LIN {X -0.205,Y -555.841,Z 989.032,A 0.000,B 0.000,C 90.000,E1 41.757} C_DIS
LIN {X 0.302,Y -553.942,Z 989.029,A 0.000,B 0.000,C 90.000,E1 41.148} C_DIS
LIN {X 0.015,Y -551.893,Z 989.026,A 0.000,B 0.000,C 90.000,E1 40.620} C_DIS
LIN {X -0.229,Y -548.482,Z 989.021,A 0.000,B 0.000,C 90.000,E1 39.806} C_DIS
LIN {X 0.068,Y -545.367,Z 989.017,A 0.000,B 0.000,C 90.000,E1 39.072} C_DIS
LIN {X -0.279,Y -542.695,Z 989.014,A 0.000,B 0.000,C 90.000,E1 38.543} C_DIS
LIN {X -0.021,Y -537.799,Z 989.008,A 0.000,B 0.000,C 90.000,E1 37.523} C_DIS
LIN {X 0.164,Y -534.006,Z 989.005,A 0.000,B 0.000,C 90.000,E1 36.790} C_DIS
LIN {X -0.018,Y -528.523,Z 988.999,A 0.000,B 0.000,C 90.000,E1 35.804} C_DIS
LIN {X -0.096,Y -523.405,Z 988.994,A 0.000,B 0.000,C 90.000,E1 34.945} C_DIS
LIN {X -0.098,Y -517.896,Z 988.989,A 0.000,B 0.000,C 90.000,E1 34.072} C_DIS
LIN {X 0.309,Y -513.063,Z 988.985,A 0.000,B 0.000,C 90.000,E1 33.293} C_DIS
LIN {X -0.136,Y -508.884,Z 988.982,A 0.000,B 0.000,C 90.000,E1 32.752} C_DIS
LIN {X 0.093,Y -504.403,Z 988.979,A 0.000,B 0.000,C 90.000,E1 32.133} C_DIS
LIN {X 0.215,Y -500.887,Z 988.976,A 0.000,B 0.000,C 90.000,E1 31.671} C_DIS
LIN {X -0.110,Y -497.223,Z 988.974,A 0.000,B 0.000,C 90.000,E1 31.258} C_DIS
LIN {X -0.112,Y -490.581,Z 988.969,A 0.000,B 0.000,C 90.000,E1 30.512} C_DIS
LIN {X 0.017,Y -485.022,Z 988.966,A 0.000,B 0.000,C 90.000,E1 29.922} C_DIS
LIN {X 0.172,Y -476.755,Z 988.962,A 0.000,B 0.000,C 90.000,E1 29.077} C_DIS
LIN {X -0.018,Y -470.857,Z 988.959,A 0.000,B 0.000,C 90.000,E1 28.537} C_DIS
LIN {X 0.163,Y -462.229,Z 988.954,A 0.000,B 0.000,C 90.000,E1 27.719} C_DIS
LIN {X -0.046,Y -451.758,Z 988.949,A 0.000,B 0.000,C 90.000,E1 26.821} C_DIS
LIN {X 0.042,Y -441.003,Z 988.944,A 0.000,B 0.000,C 90.000,E1 25.899} C_DIS
LIN {X 0.055,Y -420.137,Z 988.934,A 0.000,B 0.000,C 90.000,E1 24.027} C_DIS
LIN {X 0.018,Y -404.044,Z 988.925,A 0.000,B 0.000,C 90.000,E1 22.408} C_DIS
LIN {X -0.078,Y -399.969,Z 988.922,A 0.000,B 0.000,C 90.000,E1 21.972} C_DIS
LIN {X -0.199,Y -397.751,Z 988.921,A 0.000,B 0.000,C 90.000,E1 21.716} C_DIS
LIN {X 0.151,Y -393.382,Z 988.917,A 0.000,B 0.000,C 90.000,E1 21.046} C_DIS
LIN {X -0.105,Y -391.732,Z 988.915,A 0.000,B 0.000,C 90.000,E1 20.737} C_DIS
LIN {X 0.033,Y -390.332,Z 988.912,A 0.000,B 0.000,C 90.000,E1 20.066} C_DIS
LIN {X 0.090,Y -390.055,Z 988.908,A 0.000,B 0.000,C 90.000,E1 19.504} C_DIS
LIN {X -0.118,Y -390.561,Z 988.903,A 0.000,B 0.000,C 90.000,E1 18.471} C_DIS
LIN {X 0.071,Y -393.854,Z 988.885,A 0.000,B 0.000,C 90.000,E1 15.245} C_DIS
LIN {X 0.041,Y -398.839,Z 988.863,A 0.000,B 0.000,C 90.000,E1 11.366} C_DIS
LIN {X 0.012,Y -403.989,Z 988.846,A 0.000,B 0.000,C 90.000,E1 8.219} C_DIS
LIN {X -0.049,Y -408.655,Z 988.832,A 0.000,B 0.000,C 90.000,E1 5.796} C_DIS
LIN {X -0.025,Y -414.498,Z 988.817,A 0.000,B 0.000,C 90.000,E1 3.037} C_DIS
LIN {X 0.032,Y -417.458,Z 988.809,A 0.000,B 0.000,C 90.000,E1 1.661} C_DIS
LIN {X 0.073,Y -419.347,Z 988.806,A 0.000,B 0.000,C 90.000,E1 0.974} C_DIS
LIN {X 0.087,Y -419.875,Z 988.805,A 0.000,B 0.000,C 90.000,E1 0.802} C_DIS
LIN {X -0.145,Y -422.853,Z 988.801,A 0.000,B 0.000,C 90.000,E1 0.172} C_DIS
LIN {X 0.000,Y -423.890,Z 988.800,A 0.000,B 0.000,C 90.000,E1 360.000} C_DIS
LIN {X 0.037,Y -428.403,Z 988.797,A 0.000,B 0.000,C 90.000,E1 359.484} C_DIS
LIN {X -0.134,Y -429.256,Z 988.797,A 0.000,B 0.000,C 90.000,E1 359.427} C_DIS
LIN {X -0.068,Y -433.129,Z 988.795,A 0.000,B 0.000,C 90.000,E1 359.141} C_DIS
LIN {X -0.176,Y -441.347,Z 988.793,A 0.000,B 0.000,C 90.000,E1 358.682} C_DIS
LIN {X 0.178,Y -447.909,Z 988.791,A 0.000,B 0.000,C 90.000,E1 358.282} C_DIS
LIN {X -0.169,Y -463.031,Z 988.786,A 0.000,B 0.000,C 90.000,E1 357.478} C_DIS
LIN {X 0.080,Y -474.728,Z 988.782,A 0.000,B 0.000,C 90.000,E1 356.788} C_DIS
LIN {X 0.125,Y -487.806,Z 988.778,A 0.000,B 0.000,C 90.000,E1 356.045} C_DIS
LIN {X 0.088,Y -497.730,Z 988.775,A 0.000,B 0.000,C 90.000,E1 355.469} C_DIS
LIN {X 0.097,Y -508.908,Z 988.771,A 0.000,B 0.000,C 90.000,E1 354.780} C_DIS
LIN {X 0.239,Y -518.180,Z 988.768,A 0.000,B 0.000,C 90.000,E1 354.147} C_DIS
LIN {X -0.013,Y -524.340,Z 988.765,A 0.000,B 0.000,C 90.000,E1 353.742} C_DIS
LIN {X -0.005,Y -533.163,Z 988.761,A 0.000,B 0.000,C 90.000,E1 353.053} C_DIS
LIN {X -0.120,Y -538.896,Z 988.759,A 0.000,B 0.000,C 90.000,E1 352.591} C_DIS
LIN {X -0.208,Y -546.921,Z 988.755,A 0.000,B 0.000,C 90.000,E1 351.837} C_DIS
LIN {X -0.216,Y -552.120,Z 988.752,A 0.000,B 0.000,C 90.000,E1 351.310} C_DIS
LIN {X 0.053,Y -557.053,Z 988.749,A 0.000,B 0.000,C 90.000,E1 350.735} C_DIS
LIN {X 0.076,Y -562.660,Z 988.745,A 0.000,B 0.000,C 90.000,E1 350.038} C_DIS
LIN {X -0.162,Y -566.786,Z 988.742,A 0.000,B 0.000,C 90.000,E1 349.511} C_DIS
LIN {X 0.189,Y -570.569,Z 988.739,A 0.000,B 0.000,C 90.000,E1 348.926} C_DIS
LIN {X -0.228,Y -574.843,Z 988.735,A 0.000,B 0.000,C 90.000,E1 348.285} C_DIS
LIN {X 0.183,Y -578.041,Z 988.732,A 0.000,B 0.000,C 90.000,E1 347.701} C_DIS
LIN {X -0.056,Y -583.941,Z 988.726,A 0.000,B 0.000,C 90.000,E1 346.645} C_DIS
LIN {X -0.078,Y -589.375,Z 988.720,A 0.000,B 0.000,C 90.000,E1 345.574} C_DIS
LIN {X 0.129,Y -593.291,Z 988.715,A 0.000,B 0.000,C 90.000,E1 344.755} C_DIS
LIN {X -0.054,Y -599.436,Z 988.708,A 0.000,B 0.000,C 90.000,E1 343.449} C_DIS
LIN {X -0.221,Y -603.429,Z 988.703,A 0.000,B 0.000,C 90.000,E1 342.543} C_DIS
LIN {X -0.073,Y -608.844,Z 988.696,A 0.000,B 0.000,C 90.000,E1 341.221} C_DIS
LIN {X -0.157,Y -612.837,Z 988.690,A 0.000,B 0.000,C 90.000,E1 340.188} C_DIS
LIN {X 0.065,Y -615.611,Z 988.686,A 0.000,B 0.000,C 90.000,E1 339.390} C_DIS
LIN {X 0.045,Y -619.912,Z 988.678,A 0.000,B 0.000,C 90.000,E1 338.103} C_DIS
LIN {X -0.222,Y -621.511,Z 988.676,A 0.000,B 0.000,C 90.000,E1 337.614} C_DIS
LIN {X 0.083,Y -624.635,Z 988.670,A 0.000,B 0.000,C 90.000,E1 336.561} C_DIS
LIN {X 0.131,Y -628.204,Z 988.663,A 0.000,B 0.000,C 90.000,E1 335.281} C_DIS
LIN {X -0.046,Y -630.871,Z 988.657,A 0.000,B 0.000,C 90.000,E1 334.280} C_DIS
LIN {X 0.082,Y -633.281,Z 988.651,A 0.000,B 0.000,C 90.000,E1 333.256} C_DIS
LIN {X 0.242,Y -635.421,Z 988.646,A 0.000,B 0.000,C 90.000,E1 332.231} C_DIS
LIN {X -0.088,Y -637.969,Z 988.639,A 0.000,B 0.000,C 90.000,E1 331.001} C_DIS
LIN {X -0.015,Y -640.741,Z 988.631,A 0.000,B 0.000,C 90.000,E1 329.488} C_DIS
LIN {X -0.014,Y -642.383,Z 988.625,A 0.000,B 0.000,C 90.000,E1 328.486} C_DIS
LIN {X 0.351,Y -643.812,Z 988.619,A 0.000,B 0.000,C 90.000,E1 327.454} C_DIS
LIN {X -0.148,Y -645.119,Z 988.614,A 0.000,B 0.000,C 90.000,E1 326.501} C_DIS
LIN {X 0.204,Y -645.949,Z 988.610,A 0.000,B 0.000,C 90.000,E1 325.722} C_DIS
LIN {X 0.150,Y -647.051,Z 988.603,A 0.000,B 0.000,C 90.000,E1 324.482} C_DIS
LIN {X -0.038,Y -647.948,Z 988.596,A 0.000,B 0.000,C 90.000,E1 323.256} C_DIS
LIN {X -0.127,Y -648.450,Z 988.590,A 0.000,B 0.000,C 90.000,E1 322.271} C_DIS
LIN {X 0.062,Y -649.212,Z 988.581,A 0.000,B 0.000,C 90.000,E1 320.517} C_DIS
LIN {X -0.185,Y -649.707,Z 988.574,A 0.000,B 0.000,C 90.000,E1 319.299} C_DIS
LIN {X 0.217,Y -651.382,Z 988.559,A 0.000,B 0.000,C 90.000,E1 316.539} C_DIS
LIN {X -0.070,Y -652.394,Z 988.550,A 0.000,B 0.000,C 90.000,E1 315.081} C_DIS
LIN {X 0.052,Y -653.888,Z 988.539,A 0.000,B 0.000,C 90.000,E1 313.095} C_DIS
LIN {X 0.327,Y -654.830,Z 988.533,A 0.000,B 0.000,C 90.000,E1 311.838} C_DIS
LIN {X 0.131,Y -655.799,Z 988.524,A 0.000,B 0.000,C 90.000,E1 310.378} C_DIS
LIN {X 0.076,Y -656.458,Z 988.518,A 0.000,B 0.000,C 90.000,E1 309.152} C_DIS
LIN {X -0.064,Y -657.014,Z 988.511,A 0.000,B 0.000,C 90.000,E1 307.935} C_DIS
LIN {X -0.038,Y -657.427,Z 988.505,A 0.000,B 0.000,C 90.000,E1 306.950} C_DIS
LIN {X -0.078,Y -657.603,Z 988.501,A 0.000,B 0.000,C 90.000,E1 306.217} C_DIS
LIN {X -0.020,Y -657.818,Z 988.493,A 0.000,B 0.000,C 90.000,E1 304.739} C_DIS
LIN {X 0.219,Y -658.163,Z 988.485,A 0.000,B 0.000,C 90.000,E1 303.245} C_DIS
LIN {X -0.153,Y -664.391,Z 988.448,A 0.000,B 0.000,C 90.000,E1 296.668} C_DIS
LIN {X -0.160,Y -666.765,Z 988.440,A 0.000,B 0.000,C 90.000,E1 295.207} C_DIS
LIN {X 0.175,Y -668.283,Z 988.435,A 0.000,B 0.000,C 90.000,E1 294.207} C_DIS
LIN {X -0.080,Y -669.644,Z 988.429,A 0.000,B 0.000,C 90.000,E1 293.259} C_DIS
LIN {X 0.132,Y -670.406,Z 988.425,A 0.000,B 0.000,C 90.000,E1 292.514} C_DIS
LIN {X 0.194,Y -670.504,Z 988.422,A 0.000,B 0.000,C 90.000,E1 292.025} C_DIS
LIN {X 0.102,Y -670.488,Z 988.421,A 0.000,B 0.000,C 90.000,E1 291.791} C_DIS
LIN {X -0.209,Y -669.817,Z 988.418,A 0.000,B 0.000,C 90.000,E1 291.334} C_DIS
LIN {X -0.299,Y -669.269,Z 988.417,A 0.000,B 0.000,C 90.000,E1 291.099} C_DIS
LIN {X -0.312,Y -667.339,Z 988.415,A 0.000,B 0.000,C 90.000,E1 290.737} C_DIS
LIN {X -0.168,Y -665.582,Z 988.414,A 0.000,B 0.000,C 90.000,E1 290.482} C_DIS
LIN {X -0.099,Y -664.567,Z 988.413,A 0.000,B 0.000,C 90.000,E1 290.355} C_DIS
LIN {X -0.263,Y -663.070,Z 988.412,A 0.000,B 0.000,C 90.000,E1 290.248} C_DIS
LIN {X -0.159,Y -657.023,Z 988.410,A 0.000,B 0.000,C 90.000,E1 289.812} C_DIS
LIN {X 0.031,Y -646.511,Z 988.406,A 0.000,B 0.000,C 90.000,E1 289.141} C_DIS
LIN {X -0.299,Y -645.482,Z 988.406,A 0.000,B 0.000,C 90.000,E1 289.033} C_DIS
LIN {X -0.137,Y -645.465,Z 988.406,A 0.000,B 0.000,C 90.000,E1 289.014} C_DIS
LIN {X 0.311,Y -645.574,Z 988.405,A 0.000,B 0.000,C 90.000,E1 288.779} C_DIS
LIN {X 0.096,Y -647.600,Z 988.402,A 0.000,B 0.000,C 90.000,E1 288.362} C_DIS
LIN {X -0.194,Y -655.116,Z 988.395,A 0.000,B 0.000,C 90.000,E1 287.149} C_DIS
LIN {X 0.197,Y -657.838,Z 988.393,A 0.000,B 0.000,C 90.000,E1 286.622} C_DIS
LIN {X 0.165,Y -660.338,Z 988.390,A 0.000,B 0.000,C 90.000,E1 286.134} C_DIS
LIN {X -0.040,Y -662.472,Z 988.387,A 0.000,B 0.000,C 90.000,E1 285.662} C_DIS
LIN {X -0.229,Y -664.064,Z 988.384,A 0.000,B 0.000,C 90.000,E1 285.190} C_DIS
LIN {X -0.319,Y -664.799,Z 988.383,A 0.000,B 0.000,C 90.000,E1 284.954} C_DIS
LIN {X 0.155,Y -665.943,Z 988.380,A 0.000,B 0.000,C 90.000,E1 284.426} C_DIS
LIN {X 0.074,Y -667.201,Z 988.376,A 0.000,B 0.000,C 90.000,E1 283.703} C_DIS
LIN {X -0.237,Y -667.836,Z 988.374,A 0.000,B 0.000,C 90.000,E1 283.244} C_DIS
LIN {X 0.190,Y -668.351,Z 988.369,A 0.000,B 0.000,C 90.000,E1 282.479} C_DIS
LIN {X 0.042,Y -668.507,Z 988.367,A 0.000,B 0.000,C 90.000,E1 282.007} C_DIS
LIN {X -0.185,Y -668.277,Z 988.363,A 0.000,B 0.000,C 90.000,E1 281.299} C_DIS
LIN {X 0.188,Y -667.968,Z 988.360,A 0.000,B 0.000,C 90.000,E1 280.782} C_DIS
LIN {X 0.031,Y -667.399,Z 988.357,A 0.000,B 0.000,C 90.000,E1 280.310} C_DIS
LIN {X -0.251,Y -666.652,Z 988.355,A 0.000,B 0.000,C 90.000,E1 279.849} C_DIS
LIN {X 0.037,Y -664.846,Z 988.351,A 0.000,B 0.000,C 90.000,E1 279.095} C_DIS
LIN {X -0.151,Y -663.378,Z 988.348,A 0.000,B 0.000,C 90.000,E1 278.624} C_DIS
LIN {X 0.205,Y -661.559,Z 988.345,A 0.000,B 0.000,C 90.000,E1 278.106} C_DIS
LIN {X -0.102,Y -659.443,Z 988.342,A 0.000,B 0.000,C 90.000,E1 277.644} C_DIS
LIN {X 0.126,Y -656.103,Z 988.339,A 0.000,B 0.000,C 90.000,E1 277.011} C_DIS
LIN {X -0.140,Y -652.943,Z 988.336,A 0.000,B 0.000,C 90.000,E1 276.543} C_DIS
LIN {X 0.073,Y -649.275,Z 988.334,A 0.000,B 0.000,C 90.000,E1 276.030} C_DIS
LIN {X 0.279,Y -644.043,Z 988.330,A 0.000,B 0.000,C 90.000,E1 275.391} C_DIS
LIN {X -0.198,Y -639.512,Z 988.327,A 0.000,B 0.000,C 90.000,E1 274.935} C_DIS
LIN {X 0.069,Y -634.547,Z 988.325,A 0.000,B 0.000,C 90.000,E1 274.416} C_DIS
LIN {X -0.142,Y -627.856,Z 988.321,A 0.000,B 0.000,C 90.000,E1 273.841} C_DIS
LIN {X 0.038,Y -620.746,Z 988.318,A 0.000,B 0.000,C 90.000,E1 273.269} C_DIS
LIN {X 0.278,Y -618.053,Z 988.317,A 0.000,B 0.000,C 90.000,E1 273.037} C_DIS
LIN {X -0.294,Y -610.196,Z 988.314,A 0.000,B 0.000,C 90.000,E1 272.579} C_DIS
LIN {X -0.059,Y -603.897,Z 988.312,A 0.000,B 0.000,C 90.000,E1 272.178} C_DIS
LIN {X -0.076,Y -597.093,Z 988.310,A 0.000,B 0.000,C 90.000,E1 271.835} C_DIS
LIN {X -0.072,Y -591.854,Z 988.309,A 0.000,B 0.000,C 90.000,E1 271.604} C_DIS
LIN {X 0.033,Y -584.596,Z 988.307,A 0.000,B 0.000,C 90.000,E1 271.318} C_DIS
LIN {X -0.086,Y -576.828,Z 988.306,A 0.000,B 0.000,C 90.000,E1 271.088} C_DIS
LIN {X 0.171,Y -571.043,Z 988.305,A 0.000,B 0.000,C 90.000,E1 270.917} C_DIS
LIN {X 0.168,Y -565.048,Z 988.305,A 0.000,B 0.000,C 90.000,E1 270.802} C_DIS
LIN {X -0.005,Y -558.040,Z 988.304,A 0.000,B 0.000,C 90.000,E1 270.745} C_DIS
LIN {X -0.054,Y -543.065,Z 988.304,A 0.000,B 0.000,C 90.000,E1 270.745} C_DIS
LIN {X 0.222,Y -542.570,Z 988.302,A 0.000,B 0.000,C 90.000,E1 270.401} C_DIS
LIN {X -0.025,Y -541.364,Z 988.293,A 0.000,B 0.000,C 90.000,E1 268.740} C_DIS
LIN {X 0.103,Y -540.430,Z 988.285,A 0.000,B 0.000,C 90.000,E1 267.306} C_DIS
LIN {X -0.272,Y -538.995,Z 988.274,A 0.000,B 0.000,C 90.000,E1 265.355} C_DIS
LIN {X -0.104,Y -537.811,Z 988.266,A 0.000,B 0.000,C 90.000,E1 263.913} C_DIS
LIN {X -0.005,Y -536.805,Z 988.260,A 0.000,B 0.000,C 90.000,E1 262.761} C_DIS
LIN {X 0.146,Y -535.665,Z 988.253,A 0.000,B 0.000,C 90.000,E1 261.602} C_DIS
LIN {X -0.233,Y -533.936,Z 988.244,A 0.000,B 0.000,C 90.000,E1 259.926} C_DIS
LIN {X 0.053,Y -532.092,Z 988.234,A 0.000,B 0.000,C 90.000,E1 258.173} C_DIS
LIN {X -0.181,Y -530.829,Z 988.228,A 0.000,B 0.000,C 90.000,E1 257.048} C_DIS
LIN {X 0.159,Y -528.779,Z 988.218,A 0.000,B 0.000,C 90.000,E1 255.283} C_DIS
LIN {X 0.245,Y -526.301,Z 988.206,A 0.000,B 0.000,C 90.000,E1 252.960} C_DIS
LIN {X 0.083,Y -524.969,Z 988.199,A 0.000,B 0.000,C 90.000,E1 251.819} C_DIS
LIN {X -0.102,Y -523.557,Z 988.193,A 0.000,B 0.000,C 90.000,E1 250.678} C_DIS
LIN {X 0.175,Y -521.330,Z 988.183,A 0.000,B 0.000,C 90.000,E1 248.901} C_DIS
LIN {X -0.084,Y -519.055,Z 988.173,A 0.000,B 0.000,C 90.000,E1 247.177} C_DIS
LIN {X 0.004,Y -517.409,Z 988.167,A 0.000,B 0.000,C 90.000,E1 245.997} C_DIS
LIN {X -0.190,Y -515.692,Z 988.160,A 0.000,B 0.000,C 90.000,E1 244.845} C_DIS
LIN {X -0.279,Y -513.326,Z 988.152,A 0.000,B 0.000,C 90.000,E1 243.384} C_DIS
LIN {X 0.168,Y -511.491,Z 988.145,A 0.000,B 0.000,C 90.000,E1 242.153} C_DIS
LIN {X -0.220,Y -509.066,Z 988.137,A 0.000,B 0.000,C 90.000,E1 240.717} C_DIS
LIN {X 0.080,Y -507.515,Z 988.132,A 0.000,B 0.000,C 90.000,E1 239.793} C_DIS
LIN {X -0.130,Y -504.779,Z 988.124,A 0.000,B 0.000,C 90.000,E1 238.329} C_DIS
LIN {X -0.127,Y -501.673,Z 988.116,A 0.000,B 0.000,C 90.000,E1 236.834} C_DIS
LIN {X 0.093,Y -498.396,Z 988.107,A 0.000,B 0.000,C 90.000,E1 235.308} C_DIS
LIN {X 0.112,Y -496.271,Z 988.102,A 0.000,B 0.000,C 90.000,E1 234.402} C_DIS
LIN {X -0.182,Y -492.695,Z 988.094,A 0.000,B 0.000,C 90.000,E1 232.924} C_DIS
LIN {X -0.105,Y -488.346,Z 988.084,A 0.000,B 0.000,C 90.000,E1 231.090} C_DIS
LIN {X 0.138,Y -482.608,Z 988.070,A 0.000,B 0.000,C 90.000,E1 228.609} C_DIS
LIN {X 0.272,Y -476.521,Z 988.055,A 0.000,B 0.000,C 90.000,E1 225.810} C_DIS
LIN {X -0.001,Y -471.915,Z 988.043,A 0.000,B 0.000,C 90.000,E1 223.662} C_DIS
LIN {X 0.114,Y -468.387,Z 988.034,A 0.000,B 0.000,C 90.000,E1 222.081} C_DIS
LIN {X 0.084,Y -465.577,Z 988.027,A 0.000,B 0.000,C 90.000,E1 220.825} C_DIS
LIN {X -0.048,Y -460.589,Z 988.015,A 0.000,B 0.000,C 90.000,E1 218.624} C_DIS
LIN {X -0.049,Y -457.071,Z 988.006,A 0.000,B 0.000,C 90.000,E1 217.030} C_DIS
LIN {X 0.057,Y -452.158,Z 987.993,A 0.000,B 0.000,C 90.000,E1 214.771} C_DIS
LIN {X -0.013,Y -448.670,Z 987.984,A 0.000,B 0.000,C 90.000,E1 213.166} C_DIS
LIN {X -0.161,Y -446.535,Z 987.979,A 0.000,B 0.000,C 90.000,E1 212.212} C_DIS
LIN {X -0.156,Y -442.355,Z 987.968,A 0.000,B 0.000,C 90.000,E1 210.256} C_DIS
LIN {X -0.137,Y -438.663,Z 987.959,A 0.000,B 0.000,C 90.000,E1 208.615} C_DIS
LIN {X 0.011,Y -434.295,Z 987.948,A 0.000,B 0.000,C 90.000,E1 206.616} C_DIS
LIN {X 0.055,Y -431.318,Z 987.941,A 0.000,B 0.000,C 90.000,E1 205.283} C_DIS
LIN {X -0.181,Y -425.137,Z 987.926,A 0.000,B 0.000,C 90.000,E1 202.642} C_DIS
LIN {X 0.070,Y -420.064,Z 987.913,A 0.000,B 0.000,C 90.000,E1 200.248} C_DIS
LIN {X 0.182,Y -414.559,Z 987.897,A 0.000,B 0.000,C 90.000,E1 197.511} C_DIS
LIN {X 0.154,Y -408.961,Z 987.880,A 0.000,B 0.000,C 90.000,E1 194.426} C_DIS
LIN {X 0.026,Y -405.933,Z 987.871,A 0.000,B 0.000,C 90.000,E1 192.715} C_DIS
LIN {X 0.222,Y -403.439,Z 987.863,A 0.000,B 0.000,C 90.000,E1 191.299} C_DIS
LIN {X 0.185,Y -399.017,Z 987.849,A 0.000,B 0.000,C 90.000,E1 188.859} C_DIS
LIN {X 0.055,Y -396.649,Z 987.842,A 0.000,B 0.000,C 90.000,E1 187.473} C_DIS
LIN {X 0.001,Y -395.788,Z 987.838,A 0.000,B 0.000,C 90.000,E1 186.777} C_DIS
LIN {X -0.108,Y -395.246,Z 987.834,A 0.000,B 0.000,C 90.000,E1 186.087} C_DIS
LIN {X 0.173,Y -395.015,Z 987.829,A 0.000,B 0.000,C 90.000,E1 185.163} C_DIS
LIN {X -0.112,Y -395.395,Z 987.827,A 0.000,B 0.000,C 90.000,E1 184.821} C_DIS
LIN {X 0.172,Y -395.849,Z 987.823,A 0.000,B 0.000,C 90.000,E1 184.073} C_DIS
LIN {X 0.144,Y -397.039,Z 987.820,A 0.000,B 0.000,C 90.000,E1 183.555} C_DIS
LIN {X 0.158,Y -397.582,Z 987.819,A 0.000,B 0.000,C 90.000,E1 183.383} C_DIS
LIN {X -0.037,Y -400.045,Z 987.816,A 0.000,B 0.000,C 90.000,E1 182.808} C_DIS
LIN {X -0.064,Y -400.903,Z 987.815,A 0.000,B 0.000,C 90.000,E1 182.636} C_DIS
LIN {X -0.153,Y -405.309,Z 987.811,A 0.000,B 0.000,C 90.000,E1 181.949} C_DIS
LIN {X -0.010,Y -411.925,Z 987.806,A 0.000,B 0.000,C 90.000,E1 181.146} C_DIS
LIN {X 0.070,Y -420.445,Z 987.801,A 0.000,B 0.000,C 90.000,E1 180.229} C_DIS
LIN {X -0.103,Y -432.309,Z 987.795,A 0.000,B 0.000,C 90.000,E1 179.083} C_DIS
LIN {X 0.010,Y -439.560,Z 987.791,A 0.000,B 0.000,C 90.000,E1 178.339} C_DIS
LIN {X -0.226,Y -451.047,Z 987.784,A 0.000,B 0.000,C 90.000,E1 177.192} C_DIS
LIN {X 0.137,Y -456.691,Z 987.781,A 0.000,B 0.000,C 90.000,E1 176.560} C_DIS
LIN {X 0.060,Y -463.440,Z 987.777,A 0.000,B 0.000,C 90.000,E1 175.812} C_DIS
LIN {X -0.181,Y -470.074,Z 987.773,A 0.000,B 0.000,C 90.000,E1 175.065} C_DIS
LIN {X 0.075,Y -476.554,Z 987.768,A 0.000,B 0.000,C 90.000,E1 174.261} C_DIS
LIN {X 0.154,Y -485.042,Z 987.762,A 0.000,B 0.000,C 90.000,E1 173.166} C_DIS
LIN {X 0.189,Y -491.848,Z 987.757,A 0.000,B 0.000,C 90.000,E1 172.243} C_DIS
LIN {X 0.058,Y -499.568,Z 987.751,A 0.000,B 0.000,C 90.000,E1 171.197} C_DIS
LIN {X 0.004,Y -508.727,Z 987.744,A 0.000,B 0.000,C 90.000,E1 169.859} C_DIS
LIN {X 0.098,Y -515.688,Z 987.738,A 0.000,B 0.000,C 90.000,E1 168.814} C_DIS
LIN {X 0.074,Y -526.662,Z 987.728,A 0.000,B 0.000,C 90.000,E1 167.061} C_DIS
LIN {X -0.167,Y -535.457,Z 987.720,A 0.000,B 0.000,C 90.000,E1 165.644} C_DIS
LIN {X 0.196,Y -542.222,Z 987.714,A 0.000,B 0.000,C 90.000,E1 164.464} C_DIS
LIN {X 0.147,Y -549.582,Z 987.707,A 0.000,B 0.000,C 90.000,E1 163.196} C_DIS
LIN {X 0.207,Y -553.589,Z 987.703,A 0.000,B 0.000,C 90.000,E1 162.489} C_DIS
LIN {X -0.171,Y -562.831,Z 987.694,A 0.000,B 0.000,C 90.000,E1 160.859} C_DIS
LIN {X 0.070,Y -567.227,Z 987.689,A 0.000,B 0.000,C 90.000,E1 160.007} C_DIS
LIN {X 0.179,Y -572.904,Z 987.683,A 0.000,B 0.000,C 90.000,E1 158.901} C_DIS
LIN {X 0.295,Y -578.864,Z 987.676,A 0.000,B 0.000,C 90.000,E1 157.667} C_DIS
LIN {X -0.168,Y -585.579,Z 987.668,A 0.000,B 0.000,C 90.000,E1 156.230} C_DIS
LIN {X -0.109,Y -590.036,Z 987.662,A 0.000,B 0.000,C 90.000,E1 155.153} C_DIS
LIN {X 0.109,Y -593.130,Z 987.658,A 0.000,B 0.000,C 90.000,E1 154.332} C_DIS
LIN {X 0.271,Y -596.887,Z 987.652,A 0.000,B 0.000,C 90.000,E1 153.256} C_DIS
LIN {X -0.056,Y -600.263,Z 987.646,A 0.000,B 0.000,C 90.000,E1 152.231} C_DIS
LIN {X -0.126,Y -604.248,Z 987.638,A 0.000,B 0.000,C 90.000,E1 150.923} C_DIS
LIN {X 0.125,Y -608.863,Z 987.630,A 0.000,B 0.000,C 90.000,E1 149.331} C_DIS
LIN {X -0.097,Y -614.183,Z 987.620,A 0.000,B 0.000,C 90.000,E1 147.533} C_DIS
LIN {X -0.086,Y -620.129,Z 987.608,A 0.000,B 0.000,C 90.000,E1 145.468} C_DIS
LIN {X 0.133,Y -624.634,Z 987.600,A 0.000,B 0.000,C 90.000,E1 143.909} C_DIS
LIN {X 0.302,Y -629.794,Z 987.590,A 0.000,B 0.000,C 90.000,E1 142.110} C_DIS
LIN {X 0.212,Y -634.136,Z 987.581,A 0.000,B 0.000,C 90.000,E1 140.598} C_DIS
LIN {X -0.270,Y -637.712,Z 987.574,A 0.000,B 0.000,C 90.000,E1 139.380} C_DIS
LIN {X 0.437,Y -643.294,Z 987.563,A 0.000,B 0.000,C 90.000,E1 137.310} C_DIS
LIN {X -0.371,Y -646.952,Z 987.556,A 0.000,B 0.000,C 90.000,E1 136.134} C_DIS
LIN {X 0.004,Y -654.734,Z 987.542,A 0.000,B 0.000,C 90.000,E1 133.623} C_DIS
LIN {X -0.226,Y -661.460,Z 987.531,A 0.000,B 0.000,C 90.000,E1 131.676} C_DIS
LIN {X 0.230,Y -666.758,Z 987.523,A 0.000,B 0.000,C 90.000,E1 130.172} C_DIS
LIN {X 0.281,Y -670.105,Z 987.518,A 0.000,B 0.000,C 90.000,E1 129.197} C_DIS
LIN {X 0.072,Y -674.775,Z 987.510,A 0.000,B 0.000,C 90.000,E1 127.764} C_DIS
LIN {X 0.211,Y -677.010,Z 987.506,A 0.000,B 0.000,C 90.000,E1 127.030} C_DIS
LIN {X -0.025,Y -680.542,Z 987.499,A 0.000,B 0.000,C 90.000,E1 125.851} C_DIS
LIN {X -0.065,Y -684.007,Z 987.493,A 0.000,B 0.000,C 90.000,E1 124.659} C_DIS
LIN {X 0.139,Y -687.205,Z 987.486,A 0.000,B 0.000,C 90.000,E1 123.452} C_DIS
LIN {X 0.058,Y -691.555,Z 987.477,A 0.000,B 0.000,C 90.000,E1 121.799} C_DIS
LIN {X -0.197,Y -693.946,Z 987.471,A 0.000,B 0.000,C 90.000,E1 120.875} C_DIS
LIN {X 0.288,Y -695.542,Z 987.468,A 0.000,B 0.000,C 90.000,E1 120.129} C_DIS
LIN {X -0.170,Y -696.974,Z 987.464,A 0.000,B 0.000,C 90.000,E1 119.461} C_DIS
LIN {X 0.251,Y -698.479,Z 987.458,A 0.000,B 0.000,C 90.000,E1 118.487} C_DIS
LIN {X -0.248,Y -699.503,Z 987.453,A 0.000,B 0.000,C 90.000,E1 117.590} C_DIS
LIN {X 0.127,Y -700.716,Z 987.445,A 0.000,B 0.000,C 90.000,E1 116.155} C_DIS
LIN {X 0.010,Y -701.302,Z 987.442,A 0.000,B 0.000,C 90.000,E1 115.463} C_DIS
LIN {X -0.099,Y -701.565,Z 987.438,A 0.000,B 0.000,C 90.000,E1 114.771} C_DIS
LIN {X 0.161,Y -701.624,Z 987.435,A 0.000,B 0.000,C 90.000,E1 114.283} C_DIS
LIN {X 0.068,Y -701.284,Z 987.432,A 0.000,B 0.000,C 90.000,E1 113.823} C_DIS
LIN {X 0.060,Y -701.054,Z 987.431,A 0.000,B 0.000,C 90.000,E1 113.590} C_DIS
LIN {X -0.311,Y -700.277,Z 987.430,A 0.000,B 0.000,C 90.000,E1 113.387} C_DIS
LIN {X -0.050,Y -698.240,Z 987.427,A 0.000,B 0.000,C 90.000,E1 112.898} C_DIS
LIN {X 0.081,Y -697.376,Z 987.427,A 0.000,B 0.000,C 90.000,E1 112.770} C_DIS
LIN {X -0.245,Y -692.452,Z 987.424,A 0.000,B 0.000,C 90.000,E1 112.333} C_DIS
LIN {X -0.061,Y -690.922,Z 987.423,A 0.000,B 0.000,C 90.000,E1 112.206} C_DIS
LIN {X 0.254,Y -688.626,Z 987.423,A 0.000,B 0.000,C 90.000,E1 112.078} C_DIS
LIN {X -0.138,Y -683.905,Z 987.422,A 0.000,B 0.000,C 90.000,E1 111.950} C_DIS
LIN {X 0.102,Y -675.105,Z 987.421,A 0.000,B 0.000,C 90.000,E1 111.770} C_DIS
LIN {X 0.045,Y -673.850,Z 987.421,A 0.000,B 0.000,C 90.000,E1 111.770} C_DIS
LIN {X -0.012,Y -667.902,Z 987.421,A 0.000,B 0.000,C 90.000,E1 111.770} C_DIS
LIN {X -0.059,Y -621.920,Z 987.421,A 0.000,B 0.000,C 90.000,E1 111.770} C_DIS
LIN {X 0.073,Y -617.359,Z 987.420,A 0.000,B 0.000,C 90.000,E1 111.663} C_DIS
LIN {X 0.079,Y -610.344,Z 987.419,A 0.000,B 0.000,C 90.000,E1 111.461} C_DIS
LIN {X -0.200,Y -602.072,Z 987.417,A 0.000,B 0.000,C 90.000,E1 111.153} C_DIS
LIN {X 0.126,Y -596.157,Z 987.416,A 0.000,B 0.000,C 90.000,E1 110.791} C_DIS
LIN {X 0.059,Y -589.030,Z 987.413,A 0.000,B 0.000,C 90.000,E1 110.301} C_DIS
LIN {X 0.152,Y -577.599,Z 987.408,A 0.000,B 0.000,C 90.000,E1 109.396} C_DIS
LIN {X -0.091,Y -573.197,Z 987.406,A 0.000,B 0.000,C 90.000,E1 109.087} C_DIS
LIN {X 0.061,Y -566.709,Z 987.404,A 0.000,B 0.000,C 90.000,E1 108.671} C_DIS
LIN {X 0.110,Y -559.737,Z 987.402,A 0.000,B 0.000,C 90.000,E1 108.308} C_DIS
LIN {X -0.122,Y -551.567,Z 987.400,A 0.000,B 0.000,C 90.000,E1 107.928} C_DIS
LIN {X 0.189,Y -550.552,Z 987.399,A 0.000,B 0.000,C 90.000,E1 107.819} C_DIS
LIN {X 0.330,Y -549.468,Z 987.399,A 0.000,B 0.000,C 90.000,E1 107.692} C_DIS
LIN {X 0.281,Y -549.431,Z 987.398,A 0.000,B 0.000,C 90.000,E1 107.692} C_DIS
LIN {X 0.038,Y -548.908,Z 987.397,A 0.000,B 0.000,C 90.000,E1 107.457} C_DIS
LIN {X 0.248,Y -549.012,Z 987.393,A 0.000,B 0.000,C 90.000,E1 106.732} C_DIS
LIN {X 0.079,Y -549.759,Z 987.384,A 0.000,B 0.000,C 90.000,E1 105.064} C_DIS
LIN {X 0.006,Y -550.991,Z 987.371,A 0.000,B 0.000,C 90.000,E1 102.827} C_DIS
LIN {X 0.098,Y -553.469,Z 987.356,A 0.000,B 0.000,C 90.000,E1 100.018} C_DIS
LIN {X 0.117,Y -555.241,Z 987.346,A 0.000,B 0.000,C 90.000,E1 98.341} C_DIS
LIN {X 0.122,Y -556.702,Z 987.339,A 0.000,B 0.000,C 90.000,E1 96.947} C_DIS
LIN {X -0.053,Y -557.727,Z 987.333,A 0.000,B 0.000,C 90.000,E1 95.853} C_DIS
LIN {X -0.141,Y -558.721,Z 987.325,A 0.000,B 0.000,C 90.000,E1 94.473} C_DIS
LIN {X 0.143,Y -559.216,Z 987.320,A 0.000,B 0.000,C 90.000,E1 93.612} C_DIS
LIN {X 0.142,Y -560.123,Z 987.311,A 0.000,B 0.000,C 90.000,E1 91.949} C_DIS
LIN {X 0.160,Y -560.988,Z 987.302,A 0.000,B 0.000,C 90.000,E1 90.286} C_DIS
LIN {X 0.084,Y -561.568,Z 987.294,A 0.000,B 0.000,C 90.000,E1 88.912} C_DIS
LIN {X 0.028,Y -561.893,Z 987.286,A 0.000,B 0.000,C 90.000,E1 87.535} C_DIS
LIN {X -0.023,Y -562.093,Z 987.279,A 0.000,B 0.000,C 90.000,E1 86.159} C_DIS
LIN {X -0.035,Y -562.338,Z 987.271,A 0.000,B 0.000,C 90.000,E1 84.780} C_DIS
LIN {X 0.249,Y -562.605,Z 987.260,A 0.000,B 0.000,C 90.000,E1 82.818} C_DIS
LIN {X 0.064,Y -563.073,Z 987.250,A 0.000,B 0.000,C 90.000,E1 80.905} C_DIS
LIN {X 0.204,Y -564.039,Z 987.236,A 0.000,B 0.000,C 90.000,E1 78.409} C_DIS
LIN {X 0.209,Y -564.894,Z 987.227,A 0.000,B 0.000,C 90.000,E1 76.756} C_DIS
LIN {X 0.030,Y -566.327,Z 987.214,A 0.000,B 0.000,C 90.000,E1 74.574} C_DIS
LIN {X -0.145,Y -567.715,Z 987.204,A 0.000,B 0.000,C 90.000,E1 72.670} C_DIS
LIN {X -0.288,Y -568.864,Z 987.195,A 0.000,B 0.000,C 90.000,E1 71.040} C_DIS
LIN {X -0.216,Y -569.847,Z 987.185,A 0.000,B 0.000,C 90.000,E1 69.390} C_DIS
LIN {X 0.088,Y -570.683,Z 987.176,A 0.000,B 0.000,C 90.000,E1 67.720} C_DIS
LIN {X -0.115,Y -571.391,Z 987.167,A 0.000,B 0.000,C 90.000,E1 66.102} C_DIS
LIN {X 0.093,Y -571.888,Z 987.160,A 0.000,B 0.000,C 90.000,E1 64.717} C_DIS
LIN {X 0.134,Y -572.307,Z 987.151,A 0.000,B 0.000,C 90.000,E1 63.076} C_DIS
LIN {X 0.084,Y -572.636,Z 987.143,A 0.000,B 0.000,C 90.000,E1 61.719} C_DIS
LIN {X -0.182,Y -572.905,Z 987.135,A 0.000,B 0.000,C 90.000,E1 60.383} C_DIS
LIN {X 0.063,Y -573.130,Z 987.128,A 0.000,B 0.000,C 90.000,E1 58.997} C_DIS
LIN {X -0.187,Y -573.285,Z 987.120,A 0.000,B 0.000,C 90.000,E1 57.661} C_DIS
LIN {X -0.131,Y -573.424,Z 987.113,A 0.000,B 0.000,C 90.000,E1 56.294} C_DIS
LIN {X 0.248,Y -573.467,Z 987.105,A 0.000,B 0.000,C 90.000,E1 54.895} C_DIS
LIN {X 0.164,Y -573.198,Z 987.098,A 0.000,B 0.000,C 90.000,E1 53.543} C_DIS
LIN {X -0.067,Y -572.781,Z 987.092,A 0.000,B 0.000,C 90.000,E1 52.477} C_DIS
LIN {X 0.044,Y -572.196,Z 987.086,A 0.000,B 0.000,C 90.000,E1 51.376} C_DIS
LIN {X 0.147,Y -571.429,Z 987.079,A 0.000,B 0.000,C 90.000,E1 50.275} C_DIS
LIN {X 0.104,Y -570.722,Z 987.075,A 0.000,B 0.000,C 90.000,E1 49.461} C_DIS
LIN {X 0.048,Y -569.883,Z 987.070,A 0.000,B 0.000,C 90.000,E1 48.647} C_DIS
LIN {X 0.051,Y -568.513,Z 987.064,A 0.000,B 0.000,C 90.000,E1 47.553} C_DIS
LIN {X -0.067,Y -567.300,Z 987.060,A 0.000,B 0.000,C 90.000,E1 46.743} C_DIS
LIN {X -0.095,Y -565.379,Z 987.054,A 0.000,B 0.000,C 90.000,E1 45.648} C_DIS
LIN {X -0.239,Y -563.728,Z 987.049,A 0.000,B 0.000,C 90.000,E1 44.838} C_DIS
LIN {X 0.394,Y -561.859,Z 987.044,A 0.000,B 0.000,C 90.000,E1 43.947} C_DIS
LIN {X -0.176,Y -559.685,Z 987.040,A 0.000,B 0.000,C 90.000,E1 43.176} C_DIS
LIN {X 0.028,Y -557.264,Z 987.035,A 0.000,B 0.000,C 90.000,E1 42.324} C_DIS
LIN {X -0.211,Y -554.571,Z 987.031,A 0.000,B 0.000,C 90.000,E1 41.515} C_DIS
LIN {X -0.071,Y -551.488,Z 987.026,A 0.000,B 0.000,C 90.000,E1 40.663} C_DIS
LIN {X 0.097,Y -548.070,Z 987.021,A 0.000,B 0.000,C 90.000,E1 39.806} C_DIS
LIN {X -0.227,Y -545.598,Z 987.018,A 0.000,B 0.000,C 90.000,E1 39.277} C_DIS
LIN {X 0.037,Y -542.256,Z 987.014,A 0.000,B 0.000,C 90.000,E1 38.543} C_DIS
LIN {X -0.298,Y -536.526,Z 987.008,A 0.000,B 0.000,C 90.000,E1 37.443} C_DIS
LIN {X -0.123,Y -532.681,Z 987.004,A 0.000,B 0.000,C 90.000,E1 36.710} C_DIS
LIN {X 0.108,Y -527.082,Z 986.998,A 0.000,B 0.000,C 90.000,E1 35.678} C_DIS
LIN {X -0.154,Y -520.987,Z 986.993,A 0.000,B 0.000,C 90.000,E1 34.692} C_DIS
LIN {X 0.041,Y -513.369,Z 986.986,A 0.000,B 0.000,C 90.000,E1 33.499} C_DIS
LIN {X 0.118,Y -508.076,Z 986.982,A 0.000,B 0.000,C 90.000,E1 32.752} C_DIS
LIN {X 0.150,Y -502.426,Z 986.978,A 0.000,B 0.000,C 90.000,E1 32.005} C_DIS
LIN {X 0.215,Y -496.424,Z 986.974,A 0.000,B 0.000,C 90.000,E1 31.258} C_DIS
LIN {X -0.176,Y -490.028,Z 986.970,A 0.000,B 0.000,C 90.000,E1 30.590} C_DIS
LIN {X -0.213,Y -481.717,Z 986.965,A 0.000,B 0.000,C 90.000,E1 29.745} C_DIS
LIN {X -0.069,Y -474.566,Z 986.961,A 0.000,B 0.000,C 90.000,E1 29.027} C_DIS
LIN {X 0.055,Y -464.336,Z 986.956,A 0.000,B 0.000,C 90.000,E1 28.052} C_DIS
LIN {X 0.059,Y -453.981,Z 986.951,A 0.000,B 0.000,C 90.000,E1 27.129} C_DIS
LIN {X 0.094,Y -442.029,Z 986.945,A 0.000,B 0.000,C 90.000,E1 26.104} C_DIS
LIN {X 0.237,Y -424.254,Z 986.936,A 0.000,B 0.000,C 90.000,E1 24.515} C_DIS
LIN {X 0.006,Y -410.906,Z 986.929,A 0.000,B 0.000,C 90.000,E1 23.259} C_DIS
LIN {X 0.037,Y -400.933,Z 986.923,A 0.000,B 0.000,C 90.000,E1 22.206} C_DIS
LIN {X 0.021,Y -396.924,Z 986.921,A 0.000,B 0.000,C 90.000,E1 21.716} C_DIS
LIN {X 0.194,Y -392.996,Z 986.917,A 0.000,B 0.000,C 90.000,E1 21.099} C_DIS
LIN {X 0.147,Y -391.367,Z 986.915,A 0.000,B 0.000,C 90.000,E1 20.737} C_DIS
LIN {X -0.147,Y -390.299,Z 986.912,A 0.000,B 0.000,C 90.000,E1 20.248} C_DIS
LIN {X 0.050,Y -389.991,Z 986.909,A 0.000,B 0.000,C 90.000,E1 19.685} C_DIS
LIN {X -0.169,Y -390.848,Z 986.901,A 0.000,B 0.000,C 90.000,E1 18.236} C_DIS
LIN {X -0.015,Y -393.813,Z 986.885,A 0.000,B 0.000,C 90.000,E1 15.371} C_DIS
LIN {X 0.069,Y -398.273,Z 986.866,A 0.000,B 0.000,C 90.000,E1 11.827} C_DIS
LIN {X 0.010,Y -403.300,Z 986.848,A 0.000,B 0.000,C 90.000,E1 8.681} C_DIS
LIN {X -0.061,Y -408.519,Z 986.833,A 0.000,B 0.000,C 90.000,E1 5.910} C_DIS
LIN {X -0.042,Y -415.082,Z 986.816,A 0.000,B 0.000,C 90.000,E1 2.808} C_DIS
LIN {X 0.026,Y -418.089,Z 986.808,A 0.000,B 0.000,C 90.000,E1 1.432} C_DIS
LIN {X 0.073,Y -420.145,Z 986.804,A 0.000,B 0.000,C 90.000,E1 0.745} C_DIS
LIN {X -0.162,Y -423.020,Z 986.801,A 0.000,B 0.000,C 90.000,E1 0.115} C_DIS
LIN {X 0.161,Y -425.276,Z 986.799,A 0.000,B 0.000,C 90.000,E1 359.771} C_DIS
LIN {X 0.195,Y -428.737,Z 986.797,A 0.000,B 0.000,C 90.000,E1 359.370} C_DIS
LIN {X -0.207,Y -434.119,Z 986.794,A 0.000,B 0.000,C 90.000,E1 359.026} C_DIS
LIN {X -0.008,Y -448.089,Z 986.790,A 0.000,B 0.000,C 90.000,E1 358.224} C_DIS
LIN {X 0.006,Y -461.491,Z 986.786,A 0.000,B 0.000,C 90.000,E1 357.478} C_DIS
LIN {X 0.079,Y -471.605,Z 986.783,A 0.000,B 0.000,C 90.000,E1 356.906} C_DIS
LIN {X 0.047,Y -487.867,Z 986.778,A 0.000,B 0.000,C 90.000,E1 355.988} C_DIS
LIN {X -0.078,Y -496.093,Z 986.775,A 0.000,B 0.000,C 90.000,E1 355.527} C_DIS
LIN {X -0.081,Y -507.349,Z 986.771,A 0.000,B 0.000,C 90.000,E1 354.837} C_DIS
LIN {X -0.001,Y -515.227,Z 986.768,A 0.000,B 0.000,C 90.000,E1 354.318} C_DIS
LIN {X -0.108,Y -524.501,Z 986.765,A 0.000,B 0.000,C 90.000,E1 353.685} C_DIS
LIN {X -0.092,Y -533.277,Z 986.761,A 0.000,B 0.000,C 90.000,E1 352.996} C_DIS
LIN {X -0.128,Y -539.065,Z 986.758,A 0.000,B 0.000,C 90.000,E1 352.527} C_DIS
LIN {X 0.224,Y -547.116,Z 986.754,A 0.000,B 0.000,C 90.000,E1 351.724} C_DIS
LIN {X 0.232,Y -552.308,Z 986.751,A 0.000,B 0.000,C 90.000,E1 351.197} C_DIS
LIN {X -0.022,Y -557.218,Z 986.748,A 0.000,B 0.000,C 90.000,E1 350.679} C_DIS
LIN {X 0.260,Y -561.767,Z 986.745,A 0.000,B 0.000,C 90.000,E1 350.095} C_DIS
LIN {X -0.230,Y -566.968,Z 986.741,A 0.000,B 0.000,C 90.000,E1 349.454} C_DIS
LIN {X 0.122,Y -570.756,Z 986.738,A 0.000,B 0.000,C 90.000,E1 348.870} C_DIS
LIN {X 0.266,Y -575.062,Z 986.734,A 0.000,B 0.000,C 90.000,E1 348.173} C_DIS
LIN {X 0.114,Y -578.247,Z 986.731,A 0.000,B 0.000,C 90.000,E1 347.645} C_DIS
LIN {X 0.109,Y -583.467,Z 986.726,A 0.000,B 0.000,C 90.000,E1 346.700} C_DIS
LIN {X 0.172,Y -588.288,Z 986.721,A 0.000,B 0.000,C 90.000,E1 345.755} C_DIS
LIN {X 0.061,Y -593.577,Z 986.715,A 0.000,B 0.000,C 90.000,E1 344.700} C_DIS
LIN {X -0.183,Y -600.330,Z 986.707,A 0.000,B 0.000,C 90.000,E1 343.268} C_DIS
LIN {X 0.190,Y -604.847,Z 986.701,A 0.000,B 0.000,C 90.000,E1 342.181} C_DIS
LIN {X -0.212,Y -610.197,Z 986.694,A 0.000,B 0.000,C 90.000,E1 340.913} C_DIS
LIN {X -0.277,Y -614.125,Z 986.688,A 0.000,B 0.000,C 90.000,E1 339.880} C_DIS
LIN {X -0.071,Y -617.688,Z 986.682,A 0.000,B 0.000,C 90.000,E1 338.827} C_DIS
LIN {X -0.040,Y -621.084,Z 986.677,A 0.000,B 0.000,C 90.000,E1 337.794} C_DIS
LIN {X -0.310,Y -624.267,Z 986.671,A 0.000,B 0.000,C 90.000,E1 336.794} C_DIS
LIN {X 0.048,Y -627.897,Z 986.664,A 0.000,B 0.000,C 90.000,E1 335.485} C_DIS
LIN {X 0.134,Y -630.616,Z 986.658,A 0.000,B 0.000,C 90.000,E1 334.460} C_DIS
LIN {X -0.053,Y -632.489,Z 986.654,A 0.000,B 0.000,C 90.000,E1 333.717} C_DIS
LIN {X 0.092,Y -634.779,Z 986.648,A 0.000,B 0.000,C 90.000,E1 332.692} C_DIS
LIN {X 0.103,Y -637.883,Z 986.640,A 0.000,B 0.000,C 90.000,E1 331.179} C_DIS
LIN {X -0.244,Y -639.785,Z 986.634,A 0.000,B 0.000,C 90.000,E1 330.205} C_DIS
LIN {X -0.251,Y -641.628,Z 986.629,A 0.000,B 0.000,C 90.000,E1 329.203} C_DIS
LIN {X 0.166,Y -643.575,Z 986.622,A 0.000,B 0.000,C 90.000,E1 327.916} C_DIS
LIN {X -0.274,Y -645.262,Z 986.615,A 0.000,B 0.000,C 90.000,E1 326.707} C_DIS
LIN {X 0.137,Y -646.437,Z 986.609,A 0.000,B 0.000,C 90.000,E1 325.674} C_DIS
LIN {X 0.082,Y -647.565,Z 986.603,A 0.000,B 0.000,C 90.000,E1 324.436} C_DIS
LIN {X -0.106,Y -648.461,Z 986.596,A 0.000,B 0.000,C 90.000,E1 323.210} C_DIS
LIN {X -0.274,Y -649.024,Z 986.589,A 0.000,B 0.000,C 90.000,E1 321.984} C_DIS
LIN {X -0.095,Y -649.725,Z 986.580,A 0.000,B 0.000,C 90.000,E1 320.481} C_DIS
LIN {X 0.114,Y -650.410,Z 986.571,A 0.000,B 0.000,C 90.000,E1 318.728} C_DIS
LIN {X 0.268,Y -651.375,Z 986.563,A 0.000,B 0.000,C 90.000,E1 317.229} C_DIS
LIN {X -0.424,Y -652.263,Z 986.556,A 0.000,B 0.000,C 90.000,E1 316.053} C_DIS
LIN {X 0.275,Y -653.135,Z 986.549,A 0.000,B 0.000,C 90.000,E1 314.757} C_DIS
LIN {X -0.063,Y -654.702,Z 986.538,A 0.000,B 0.000,C 90.000,E1 312.813} C_DIS
LIN {X -0.186,Y -655.419,Z 986.532,A 0.000,B 0.000,C 90.000,E1 311.838} C_DIS
LIN {X 0.131,Y -656.410,Z 986.524,A 0.000,B 0.000,C 90.000,E1 310.334} C_DIS
LIN {X 0.045,Y -656.958,Z 986.519,A 0.000,B 0.000,C 90.000,E1 309.358} C_DIS
LIN {X -0.027,Y -657.648,Z 986.511,A 0.000,B 0.000,C 90.000,E1 307.890} C_DIS
LIN {X 0.411,Y -658.084,Z 986.505,A 0.000,B 0.000,C 90.000,E1 306.870} C_DIS
LIN {X -0.014,Y -658.245,Z 986.501,A 0.000,B 0.000,C 90.000,E1 306.171} C_DIS
LIN {X -0.006,Y -658.543,Z 986.491,A 0.000,B 0.000,C 90.000,E1 304.452} C_DIS
LIN {X 0.070,Y -659.804,Z 986.474,A 0.000,B 0.000,C 90.000,E1 301.258} C_DIS
LIN {X -0.239,Y -666.678,Z 986.443,A 0.000,B 0.000,C 90.000,E1 295.668} C_DIS
LIN {X 0.379,Y -668.262,Z 986.437,A 0.000,B 0.000,C 90.000,E1 294.643} C_DIS
LIN {X 0.016,Y -670.085,Z 986.430,A 0.000,B 0.000,C 90.000,E1 293.462} C_DIS
LIN {X 0.337,Y -670.731,Z 986.428,A 0.000,B 0.000,C 90.000,E1 292.950} C_DIS
LIN {X -0.219,Y -671.189,Z 986.425,A 0.000,B 0.000,C 90.000,E1 292.514} C_DIS
LIN {X 0.008,Y -671.239,Z 986.421,A 0.000,B 0.000,C 90.000,E1 291.770} C_DIS
LIN {X 0.076,Y -670.506,Z 986.418,A 0.000,B 0.000,C 90.000,E1 291.280} C_DIS
LIN {X -0.011,Y -669.944,Z 986.417,A 0.000,B 0.000,C 90.000,E1 291.046} C_DIS
LIN {X 0.066,Y -669.334,Z 986.416,A 0.000,B 0.000,C 90.000,E1 290.918} C_DIS
LIN {X 0.216,Y -667.669,Z 986.415,A 0.000,B 0.000,C 90.000,E1 290.663} C_DIS
LIN {X 0.125,Y -665.878,Z 986.414,A 0.000,B 0.000,C 90.000,E1 290.429} C_DIS
LIN {X 0.194,Y -664.817,Z 986.413,A 0.000,B 0.000,C 90.000,E1 290.301} C_DIS
LIN {X 0.097,Y -661.514,Z 986.412,A 0.000,B 0.000,C 90.000,E1 290.066} C_DIS
LIN {X 0.300,Y -657.326,Z 986.410,A 0.000,B 0.000,C 90.000,E1 289.758} C_DIS
LIN {X 0.140,Y -652.762,Z 986.408,A 0.000,B 0.000,C 90.000,E1 289.504} C_DIS
LIN {X -0.104,Y -647.001,Z 986.406,A 0.000,B 0.000,C 90.000,E1 289.141} C_DIS
LIN {X 0.069,Y -646.329,Z 986.406,A 0.000,B 0.000,C 90.000,E1 289.033} C_DIS
LIN {X 0.034,Y -646.328,Z 986.406,A 0.000,B 0.000,C 90.000,E1 289.033} C_DIS
LIN {X 0.081,Y -646.521,Z 986.405,A 0.000,B 0.000,C 90.000,E1 288.852} C_DIS
LIN {X 0.019,Y -649.569,Z 986.401,A 0.000,B 0.000,C 90.000,E1 288.236} C_DIS
LIN {X 0.030,Y -654.746,Z 986.397,A 0.000,B 0.000,C 90.000,E1 287.402} C_DIS
LIN {X -0.017,Y -657.608,Z 986.394,A 0.000,B 0.000,C 90.000,E1 286.913} C_DIS
LIN {X -0.198,Y -660.865,Z 986.391,A 0.000,B 0.000,C 90.000,E1 286.315} C_DIS
LIN {X 0.239,Y -663.012,Z 986.388,A 0.000,B 0.000,C 90.000,E1 285.788} C_DIS
LIN {X 0.146,Y -663.991,Z 986.387,A 0.000,B 0.000,C 90.000,E1 285.552} C_DIS
LIN {X 0.143,Y -665.500,Z 986.384,A 0.000,B 0.000,C 90.000,E1 285.064} C_DIS
LIN {X -0.107,Y -667.275,Z 986.380,A 0.000,B 0.000,C 90.000,E1 284.356} C_DIS
LIN {X 0.309,Y -668.432,Z 986.376,A 0.000,B 0.000,C 90.000,E1 283.592} C_DIS
LIN {X 0.161,Y -669.050,Z 986.373,A 0.000,B 0.000,C 90.000,E1 283.119} C_DIS
LIN {X -0.056,Y -669.517,Z 986.369,A 0.000,B 0.000,C 90.000,E1 282.411} C_DIS
LIN {X -0.341,Y -669.628,Z 986.366,A 0.000,B 0.000,C 90.000,E1 281.951} C_DIS
LIN {X 0.101,Y -669.388,Z 986.362,A 0.000,B 0.000,C 90.000,E1 281.186} C_DIS
LIN {X 0.028,Y -669.279,Z 986.361,A 0.000,B 0.000,C 90.000,E1 280.950} C_DIS
LIN {X -0.322,Y -668.436,Z 986.357,A 0.000,B 0.000,C 90.000,E1 280.254} C_DIS
LIN {X 0.175,Y -667.646,Z 986.354,A 0.000,B 0.000,C 90.000,E1 279.726} C_DIS
LIN {X -0.103,Y -666.510,Z 986.351,A 0.000,B 0.000,C 90.000,E1 279.265} C_DIS
LIN {X 0.274,Y -665.120,Z 986.349,A 0.000,B 0.000,C 90.000,E1 278.746} C_DIS
LIN {X 0.084,Y -663.383,Z 986.346,A 0.000,B 0.000,C 90.000,E1 278.276} C_DIS
LIN {X -0.215,Y -661.362,Z 986.343,A 0.000,B 0.000,C 90.000,E1 277.814} C_DIS
LIN {X 0.243,Y -660.262,Z 986.342,A 0.000,B 0.000,C 90.000,E1 277.530} C_DIS
LIN {X -0.071,Y -657.636,Z 986.339,A 0.000,B 0.000,C 90.000,E1 277.068} C_DIS
LIN {X 0.216,Y -653.670,Z 986.336,A 0.000,B 0.000,C 90.000,E1 276.429} C_DIS
LIN {X -0.144,Y -650.001,Z 986.333,A 0.000,B 0.000,C 90.000,E1 275.967} C_DIS
LIN {X 0.001,Y -644.751,Z 986.330,A 0.000,B 0.000,C 90.000,E1 275.334} C_DIS
LIN {X 0.170,Y -640.208,Z 986.327,A 0.000,B 0.000,C 90.000,E1 274.821} C_DIS
LIN {X -0.196,Y -635.270,Z 986.324,A 0.000,B 0.000,C 90.000,E1 274.359} C_DIS
LIN {X -0.164,Y -628.822,Z 986.321,A 0.000,B 0.000,C 90.000,E1 273.784} C_DIS
LIN {X -0.080,Y -623.196,Z 986.318,A 0.000,B 0.000,C 90.000,E1 273.326} C_DIS
LIN {X 0.183,Y -619.006,Z 986.317,A 0.000,B 0.000,C 90.000,E1 272.980} C_DIS
LIN {X 0.230,Y -611.377,Z 986.314,A 0.000,B 0.000,C 90.000,E1 272.465} C_DIS
LIN {X -0.191,Y -605.030,Z 986.312,A 0.000,B 0.000,C 90.000,E1 272.121} C_DIS
LIN {X -0.194,Y -598.348,Z 986.310,A 0.000,B 0.000,C 90.000,E1 271.776} C_DIS
LIN {X 0.176,Y -591.413,Z 986.308,A 0.000,B 0.000,C 90.000,E1 271.432} C_DIS
LIN {X -0.203,Y -584.396,Z 986.307,A 0.000,B 0.000,C 90.000,E1 271.203} C_DIS
LIN {X -0.215,Y -576.978,Z 986.305,A 0.000,B 0.000,C 90.000,E1 270.974} C_DIS
LIN {X 0.050,Y -571.141,Z 986.305,A 0.000,B 0.000,C 90.000,E1 270.802} C_DIS
LIN {X -0.031,Y -564.909,Z 986.304,A 0.000,B 0.000,C 90.000,E1 270.688} C_DIS
LIN {X -0.192,Y -557.686,Z 986.303,A 0.000,B 0.000,C 90.000,E1 270.630} C_DIS
LIN {X -0.242,Y -543.806,Z 986.303,A 0.000,B 0.000,C 90.000,E1 270.630} C_DIS
LIN {X -0.206,Y -543.017,Z 986.303,A 0.000,B 0.000,C 90.000,E1 270.573} C_DIS
LIN {X -0.238,Y -542.971,Z 986.303,A 0.000,B 0.000,C 90.000,E1 270.573} C_DIS
LIN {X -0.076,Y -542.459,Z 986.301,A 0.000,B 0.000,C 90.000,E1 270.172} C_DIS
LIN {X 0.085,Y -541.274,Z 986.292,A 0.000,B 0.000,C 90.000,E1 268.453} C_DIS
LIN {X 0.190,Y -540.525,Z 986.285,A 0.000,B 0.000,C 90.000,E1 267.306} C_DIS
LIN {X -0.182,Y -539.098,Z 986.274,A 0.000,B 0.000,C 90.000,E1 265.355} C_DIS
LIN {X -0.012,Y -537.964,Z 986.266,A 0.000,B 0.000,C 90.000,E1 263.913} C_DIS
LIN {X 0.089,Y -536.922,Z 986.260,A 0.000,B 0.000,C 90.000,E1 262.761} C_DIS
LIN {X 0.241,Y -535.801,Z 986.254,A 0.000,B 0.000,C 90.000,E1 261.602} C_DIS
LIN {X -0.096,Y -534.366,Z 986.246,A 0.000,B 0.000,C 90.000,E1 260.208} C_DIS
LIN {X 0.108,Y -532.544,Z 986.236,A 0.000,B 0.000,C 90.000,E1 258.465} C_DIS
LIN {X -0.197,Y -530.947,Z 986.228,A 0.000,B 0.000,C 90.000,E1 257.061} C_DIS
LIN {X 0.262,Y -528.882,Z 986.218,A 0.000,B 0.000,C 90.000,E1 255.283} C_DIS
LIN {X -0.152,Y -526.413,Z 986.206,A 0.000,B 0.000,C 90.000,E1 253.015} C_DIS
LIN {X 0.190,Y -525.084,Z 986.199,A 0.000,B 0.000,C 90.000,E1 251.819} C_DIS
LIN {X 0.168,Y -523.277,Z 986.191,A 0.000,B 0.000,C 90.000,E1 250.369} C_DIS
LIN {X -0.201,Y -521.438,Z 986.183,A 0.000,B 0.000,C 90.000,E1 248.954} C_DIS
LIN {X 0.028,Y -519.176,Z 986.173,A 0.000,B 0.000,C 90.000,E1 247.177} C_DIS
LIN {X -0.020,Y -517.971,Z 986.168,A 0.000,B 0.000,C 90.000,E1 246.305} C_DIS
LIN {X -0.074,Y -515.790,Z 986.160,A 0.000,B 0.000,C 90.000,E1 244.845} C_DIS
LIN {X -0.163,Y -513.427,Z 986.152,A 0.000,B 0.000,C 90.000,E1 243.384} C_DIS
LIN {X 0.285,Y -511.595,Z 986.146,A 0.000,B 0.000,C 90.000,E1 242.153} C_DIS
LIN {X -0.101,Y -509.170,Z 986.137,A 0.000,B 0.000,C 90.000,E1 240.717} C_DIS
LIN {X -0.167,Y -507.072,Z 986.131,A 0.000,B 0.000,C 90.000,E1 239.537} C_DIS
LIN {X -0.008,Y -504.881,Z 986.124,A 0.000,B 0.000,C 90.000,E1 238.329} C_DIS
LIN {X -0.006,Y -501.765,Z 986.116,A 0.000,B 0.000,C 90.000,E1 236.834} C_DIS
LIN {X 0.215,Y -498.472,Z 986.107,A 0.000,B 0.000,C 90.000,E1 235.308} C_DIS
LIN {X -0.033,Y -494.985,Z 986.099,A 0.000,B 0.000,C 90.000,E1 233.829} C_DIS
LIN {X -0.203,Y -492.049,Z 986.092,A 0.000,B 0.000,C 90.000,E1 232.637} C_DIS
LIN {X 0.022,Y -488.482,Z 986.084,A 0.000,B 0.000,C 90.000,E1 231.090} C_DIS
LIN {X 0.133,Y -483.435,Z 986.072,A 0.000,B 0.000,C 90.000,E1 228.933} C_DIS
LIN {X 0.291,Y -477.273,Z 986.057,A 0.000,B 0.000,C 90.000,E1 226.134} C_DIS
LIN {X 0.265,Y -473.323,Z 986.046,A 0.000,B 0.000,C 90.000,E1 224.271} C_DIS
LIN {X -0.028,Y -470.597,Z 986.039,A 0.000,B 0.000,C 90.000,E1 223.056} C_DIS
LIN {X 0.155,Y -466.397,Z 986.029,A 0.000,B 0.000,C 90.000,E1 221.148} C_DIS
LIN {X -0.058,Y -462.119,Z 986.018,A 0.000,B 0.000,C 90.000,E1 219.277} C_DIS
LIN {X -0.014,Y -457.889,Z 986.008,A 0.000,B 0.000,C 90.000,E1 217.363} C_DIS
LIN {X 0.012,Y -453.662,Z 985.997,A 0.000,B 0.000,C 90.000,E1 215.438} C_DIS
LIN {X -0.035,Y -450.159,Z 985.988,A 0.000,B 0.000,C 90.000,E1 213.833} C_DIS
LIN {X -0.094,Y -447.375,Z 985.981,A 0.000,B 0.000,C 90.000,E1 212.546} C_DIS
LIN {X -0.016,Y -442.448,Z 985.968,A 0.000,B 0.000,C 90.000,E1 210.256} C_DIS
LIN {X -0.036,Y -439.523,Z 985.961,A 0.000,B 0.000,C 90.000,E1 208.949} C_DIS
LIN {X 0.155,Y -434.392,Z 985.948,A 0.000,B 0.000,C 90.000,E1 206.616} C_DIS
LIN {X -0.007,Y -432.209,Z 985.943,A 0.000,B 0.000,C 90.000,E1 205.643} C_DIS
LIN {X 0.000,Y -427.528,Z 985.931,A 0.000,B 0.000,C 90.000,E1 203.643} C_DIS
LIN {X -0.051,Y -423.765,Z 985.922,A 0.000,B 0.000,C 90.000,E1 201.972} C_DIS
LIN {X -0.176,Y -420.188,Z 985.913,A 0.000,B 0.000,C 90.000,E1 200.301} C_DIS
LIN {X -0.189,Y -414.638,Z 985.898,A 0.000,B 0.000,C 90.000,E1 197.583} C_DIS
LIN {X -0.110,Y -409.640,Z 985.882,A 0.000,B 0.000,C 90.000,E1 194.828} C_DIS
LIN {X 0.152,Y -407.171,Z 985.875,A 0.000,B 0.000,C 90.000,E1 193.411} C_DIS
LIN {X -0.114,Y -404.730,Z 985.867,A 0.000,B 0.000,C 90.000,E1 192.063} C_DIS
LIN {X -0.031,Y -400.826,Z 985.855,A 0.000,B 0.000,C 90.000,E1 189.962} C_DIS
LIN {X -0.193,Y -396.546,Z 985.842,A 0.000,B 0.000,C 90.000,E1 187.530} C_DIS
LIN {X 0.114,Y -395.232,Z 985.836,A 0.000,B 0.000,C 90.000,E1 186.429} C_DIS
LIN {X -0.001,Y -394.573,Z 985.832,A 0.000,B 0.000,C 90.000,E1 185.739} C_DIS
LIN {X -0.118,Y -394.380,Z 985.828,A 0.000,B 0.000,C 90.000,E1 185.049} C_DIS
LIN {X 0.156,Y -394.634,Z 985.824,A 0.000,B 0.000,C 90.000,E1 184.302} C_DIS
LIN {X 0.110,Y -395.053,Z 985.822,A 0.000,B 0.000,C 90.000,E1 183.955} C_DIS
LIN {X 0.036,Y -395.657,Z 985.820,A 0.000,B 0.000,C 90.000,E1 183.612} C_DIS
LIN {X 0.044,Y -396.484,Z 985.818,A 0.000,B 0.000,C 90.000,E1 183.269} C_DIS
LIN {X -0.033,Y -398.523,Z 985.815,A 0.000,B 0.000,C 90.000,E1 182.751} C_DIS
LIN {X -0.090,Y -400.033,Z 985.813,A 0.000,B 0.000,C 90.000,E1 182.407} C_DIS
LIN {X -0.140,Y -402.844,Z 985.811,A 0.000,B 0.000,C 90.000,E1 181.949} C_DIS
LIN {X -0.172,Y -405.252,Z 985.809,A 0.000,B 0.000,C 90.000,E1 181.604} C_DIS
LIN {X 0.087,Y -411.882,Z 985.805,A 0.000,B 0.000,C 90.000,E1 180.802} C_DIS
LIN {X 0.158,Y -420.616,Z 985.800,A 0.000,B 0.000,C 90.000,E1 179.885} C_DIS
LIN {X -0.159,Y -431.062,Z 985.794,A 0.000,B 0.000,C 90.000,E1 178.912} C_DIS
LIN {X 0.171,Y -438.133,Z 985.790,A 0.000,B 0.000,C 90.000,E1 178.167} C_DIS
LIN {X 0.013,Y -446.798,Z 985.785,A 0.000,B 0.000,C 90.000,E1 177.306} C_DIS
LIN {X -0.148,Y -455.336,Z 985.780,A 0.000,B 0.000,C 90.000,E1 176.445} C_DIS
LIN {X 0.120,Y -463.295,Z 985.775,A 0.000,B 0.000,C 90.000,E1 175.527} C_DIS
LIN {X 0.047,Y -471.254,Z 985.770,A 0.000,B 0.000,C 90.000,E1 174.609} C_DIS
LIN {X 0.112,Y -476.521,Z 985.767,A 0.000,B 0.000,C 90.000,E1 173.976} C_DIS
LIN {X 0.144,Y -483.825,Z 985.762,A 0.000,B 0.000,C 90.000,E1 173.053} C_DIS
LIN {X 0.134,Y -492.816,Z 985.755,A 0.000,B 0.000,C 90.000,E1 171.837} C_DIS
LIN {X -0.223,Y -499.530,Z 985.750,A 0.000,B 0.000,C 90.000,E1 170.971} C_DIS
LIN {X 0.177,Y -508.735,Z 985.742,A 0.000,B 0.000,C 90.000,E1 169.577} C_DIS
LIN {X -0.115,Y -515.616,Z 985.737,A 0.000,B 0.000,C 90.000,E1 168.578} C_DIS
LIN {X 0.165,Y -525.820,Z 985.728,A 0.000,B 0.000,C 90.000,E1 166.937} C_DIS
LIN {X -0.082,Y -534.606,Z 985.720,A 0.000,B 0.000,C 90.000,E1 165.519} C_DIS
LIN {X -0.248,Y -541.399,Z 985.713,A 0.000,B 0.000,C 90.000,E1 164.393} C_DIS
LIN {X 0.059,Y -548.800,Z 985.706,A 0.000,B 0.000,C 90.000,E1 163.087} C_DIS
LIN {X 0.145,Y -553.607,Z 985.701,A 0.000,B 0.000,C 90.000,E1 162.236} C_DIS
LIN {X -0.114,Y -562.071,Z 985.693,A 0.000,B 0.000,C 90.000,E1 160.732} C_DIS
LIN {X 0.224,Y -565.893,Z 985.689,A 0.000,B 0.000,C 90.000,E1 160.007} C_DIS
LIN {X -0.032,Y -570.169,Z 985.685,A 0.000,B 0.000,C 90.000,E1 159.209} C_DIS
LIN {X 0.137,Y -572.962,Z 985.682,A 0.000,B 0.000,C 90.000,E1 158.646} C_DIS
LIN {X -0.123,Y -577.667,Z 985.676,A 0.000,B 0.000,C 90.000,E1 157.720} C_DIS
LIN {X -0.004,Y -583.813,Z 985.669,A 0.000,B 0.000,C 90.000,E1 156.357} C_DIS
LIN {X 0.032,Y -588.403,Z 985.663,A 0.000,B 0.000,C 90.000,E1 155.281} C_DIS
LIN {X 0.341,Y -590.598,Z 985.660,A 0.000,B 0.000,C 90.000,E1 154.717} C_DIS
LIN {X 0.132,Y -592.642,Z 985.657,A 0.000,B 0.000,C 90.000,E1 154.204} C_DIS
LIN {X -0.156,Y -595.487,Z 985.652,A 0.000,B 0.000,C 90.000,E1 153.435} C_DIS
LIN {X -0.049,Y -599.770,Z 985.645,A 0.000,B 0.000,C 90.000,E1 152.103} C_DIS
LIN {X 0.013,Y -602.231,Z 985.641,A 0.000,B 0.000,C 90.000,E1 151.307} C_DIS
LIN {X 0.169,Y -607.641,Z 985.630,A 0.000,B 0.000,C 90.000,E1 149.459} C_DIS
LIN {X -0.077,Y -613.032,Z 985.620,A 0.000,B 0.000,C 90.000,E1 147.661} C_DIS
LIN {X -0.090,Y -619.073,Z 985.609,A 0.000,B 0.000,C 90.000,E1 145.595} C_DIS
LIN {X 0.112,Y -623.623,Z 985.600,A 0.000,B 0.000,C 90.000,E1 144.036} C_DIS
LIN {X -0.120,Y -628.844,Z 985.590,A 0.000,B 0.000,C 90.000,E1 142.271} C_DIS
LIN {X 0.043,Y -633.943,Z 985.581,A 0.000,B 0.000,C 90.000,E1 140.481} C_DIS
LIN {X 0.052,Y -637.531,Z 985.573,A 0.000,B 0.000,C 90.000,E1 139.218} C_DIS
LIN {X -0.147,Y -643.181,Z 985.562,A 0.000,B 0.000,C 90.000,E1 137.229} C_DIS
LIN {X -0.045,Y -646.870,Z 985.555,A 0.000,B 0.000,C 90.000,E1 135.972} C_DIS
LIN {X 0.423,Y -653.153,Z 985.544,A 0.000,B 0.000,C 90.000,E1 133.947} C_DIS
LIN {X 0.132,Y -660.698,Z 985.532,A 0.000,B 0.000,C 90.000,E1 131.757} C_DIS
LIN {X 0.070,Y -666.038,Z 985.524,A 0.000,B 0.000,C 90.000,E1 130.297} C_DIS
LIN {X -0.326,Y -670.252,Z 985.517,A 0.000,B 0.000,C 90.000,E1 129.116} C_DIS
LIN {X -0.126,Y -674.218,Z 985.510,A 0.000,B 0.000,C 90.000,E1 127.890} C_DIS
LIN {X 0.005,Y -677.183,Z 985.505,A 0.000,B 0.000,C 90.000,E1 126.916} C_DIS
LIN {X -0.089,Y -680.716,Z 985.498,A 0.000,B 0.000,C 90.000,E1 125.724} C_DIS
LIN {X -0.122,Y -684.205,Z 985.492,A 0.000,B 0.000,C 90.000,E1 124.532} C_DIS
LIN {X 0.468,Y -687.417,Z 985.485,A 0.000,B 0.000,C 90.000,E1 123.293} C_DIS
LIN {X 0.017,Y -691.758,Z 985.476,A 0.000,B 0.000,C 90.000,E1 121.671} C_DIS
LIN {X -0.470,Y -693.562,Z 985.472,A 0.000,B 0.000,C 90.000,E1 121.003} C_DIS
LIN {X 0.254,Y -695.664,Z 985.467,A 0.000,B 0.000,C 90.000,E1 120.001} C_DIS
LIN {X 0.152,Y -696.658,Z 985.464,A 0.000,B 0.000,C 90.000,E1 119.539} C_DIS
LIN {X -0.039,Y -698.182,Z 985.459,A 0.000,B 0.000,C 90.000,E1 118.615} C_DIS
LIN {X 0.135,Y -699.005,Z 985.455,A 0.000,B 0.000,C 90.000,E1 117.897} C_DIS
LIN {X 0.182,Y -700.270,Z 985.447,A 0.000,B 0.000,C 90.000,E1 116.488} C_DIS
LIN {X -0.020,Y -701.190,Z 985.441,A 0.000,B 0.000,C 90.000,E1 115.335} C_DIS
LIN {X -0.131,Y -701.407,Z 985.437,A 0.000,B 0.000,C 90.000,E1 114.643} C_DIS
LIN {X 0.129,Y -701.416,Z 985.434,A 0.000,B 0.000,C 90.000,E1 114.155} C_DIS
LIN {X 0.034,Y -700.994,Z 985.432,A 0.000,B 0.000,C 90.000,E1 113.695} C_DIS
LIN {X 0.025,Y -700.482,Z 985.430,A 0.000,B 0.000,C 90.000,E1 113.462} C_DIS
LIN {X -0.082,Y -698.649,Z 985.428,A 0.000,B 0.000,C 90.000,E1 113.003} C_DIS
LIN {X -0.222,Y -698.047,Z 985.427,A 0.000,B 0.000,C 90.000,E1 112.898} C_DIS
LIN {X -0.091,Y -697.134,Z 985.427,A 0.000,B 0.000,C 90.000,E1 112.770} C_DIS
LIN {X 0.192,Y -692.221,Z 985.424,A 0.000,B 0.000,C 90.000,E1 112.280} C_DIS
LIN {X -0.275,Y -690.562,Z 985.423,A 0.000,B 0.000,C 90.000,E1 112.206} C_DIS
LIN {X -0.263,Y -685.896,Z 985.422,A 0.000,B 0.000,C 90.000,E1 112.025} C_DIS
LIN {X -0.168,Y -683.737,Z 985.422,A 0.000,B 0.000,C 90.000,E1 111.950} C_DIS
LIN {X 0.120,Y -675.655,Z 985.421,A 0.000,B 0.000,C 90.000,E1 111.770} C_DIS
LIN {X -0.042,Y -672.266,Z 985.421,A 0.000,B 0.000,C 90.000,E1 111.770} C_DIS
LIN {X -0.095,Y -668.262,Z 985.421,A 0.000,B 0.000,C 90.000,E1 111.770} C_DIS
LIN {X -0.132,Y -622.522,Z 985.421,A 0.000,B 0.000,C 90.000,E1 111.770} C_DIS
LIN {X -0.084,Y -616.593,Z 985.420,A 0.000,B 0.000,C 90.000,E1 111.642} C_DIS
LIN {X -0.227,Y -610.085,Z 985.419,A 0.000,B 0.000,C 90.000,E1 111.461} C_DIS
LIN {X 0.021,Y -601.907,Z 985.417,A 0.000,B 0.000,C 90.000,E1 111.099} C_DIS
LIN {X -0.051,Y -597.466,Z 985.416,A 0.000,B 0.000,C 90.000,E1 110.865} C_DIS
LIN {X 0.119,Y -591.114,Z 985.414,A 0.000,B 0.000,C 90.000,E1 110.429} C_DIS
LIN {X -0.024,Y -577.628,Z 985.408,A 0.000,B 0.000,C 90.000,E1 109.396} C_DIS
LIN {X -0.291,Y -573.148,Z 985.406,A 0.000,B 0.000,C 90.000,E1 109.087} C_DIS
LIN {X -0.193,Y -566.572,Z 985.404,A 0.000,B 0.000,C 90.000,E1 108.671} C_DIS
LIN {X 0.247,Y -551.685,Z 985.399,A 0.000,B 0.000,C 90.000,E1 107.873} C_DIS
LIN {X 0.154,Y -549.512,Z 985.398,A 0.000,B 0.000,C 90.000,E1 107.692} C_DIS
LIN {X 0.116,Y -549.490,Z 985.398,A 0.000,B 0.000,C 90.000,E1 107.692} C_DIS
LIN {X 0.173,Y -549.003,Z 985.397,A 0.000,B 0.000,C 90.000,E1 107.457} C_DIS
LIN {X 0.088,Y -549.155,Z 985.392,A 0.000,B 0.000,C 90.000,E1 106.622} C_DIS
LIN {X -0.070,Y -549.887,Z 985.383,A 0.000,B 0.000,C 90.000,E1 104.954} C_DIS
LIN {X -0.091,Y -552.047,Z 985.364,A 0.000,B 0.000,C 90.000,E1 101.591} C_DIS
LIN {X 0.101,Y -553.939,Z 985.354,A 0.000,B 0.000,C 90.000,E1 99.613} C_DIS
LIN {X 0.088,Y -555.426,Z 985.346,A 0.000,B 0.000,C 90.000,E1 98.219} C_DIS
LIN {X 0.019,Y -556.850,Z 985.338,A 0.000,B 0.000,C 90.000,E1 96.834} C_DIS
LIN {X -0.153,Y -557.820,Z 985.332,A 0.000,B 0.000,C 90.000,E1 95.739} C_DIS
LIN {X -0.235,Y -558.799,Z 985.324,A 0.000,B 0.000,C 90.000,E1 94.359} C_DIS
LIN {X 0.253,Y -559.617,Z 985.316,A 0.000,B 0.000,C 90.000,E1 92.922} C_DIS
LIN {X 0.162,Y -560.343,Z 985.309,A 0.000,B 0.000,C 90.000,E1 91.547} C_DIS
LIN {X -0.023,Y -560.916,Z 985.303,A 0.000,B 0.000,C 90.000,E1 90.458} C_DIS
LIN {X -0.198,Y -561.406,Z 985.296,A 0.000,B 0.000,C 90.000,E1 89.370} C_DIS
LIN {X 0.191,Y -561.751,Z 985.290,A 0.000,B 0.000,C 90.000,E1 88.224} C_DIS
LIN {X 0.261,Y -562.080,Z 985.281,A 0.000,B 0.000,C 90.000,E1 86.560} C_DIS
LIN {X -0.215,Y -562.319,Z 985.272,A 0.000,B 0.000,C 90.000,E1 84.951} C_DIS
LIN {X 0.006,Y -562.583,Z 985.261,A 0.000,B 0.000,C 90.000,E1 82.996} C_DIS
LIN {X -0.191,Y -563.023,Z 985.250,A 0.000,B 0.000,C 90.000,E1 81.084} C_DIS
LIN {X 0.048,Y -563.969,Z 985.237,A 0.000,B 0.000,C 90.000,E1 78.578} C_DIS
LIN {X 0.098,Y -564.951,Z 985.226,A 0.000,B 0.000,C 90.000,E1 76.645} C_DIS
LIN {X -0.253,Y -566.236,Z 985.215,A 0.000,B 0.000,C 90.000,E1 74.755} C_DIS
LIN {X 0.277,Y -567.599,Z 985.205,A 0.000,B 0.000,C 90.000,E1 72.779} C_DIS
LIN {X -0.197,Y -568.550,Z 985.197,A 0.000,B 0.000,C 90.000,E1 71.456} C_DIS
LIN {X 0.064,Y -569.421,Z 985.189,A 0.000,B 0.000,C 90.000,E1 70.061} C_DIS
LIN {X 0.150,Y -570.316,Z 985.180,A 0.000,B 0.000,C 90.000,E1 68.411} C_DIS
LIN {X -0.246,Y -570.814,Z 985.174,A 0.000,B 0.000,C 90.000,E1 67.358} C_DIS
LIN {X -0.053,Y -571.359,Z 985.167,A 0.000,B 0.000,C 90.000,E1 65.973} C_DIS
LIN {X 0.154,Y -571.841,Z 985.159,A 0.000,B 0.000,C 90.000,E1 64.588} C_DIS
LIN {X -0.151,Y -572.214,Z 985.151,A 0.000,B 0.000,C 90.000,E1 63.256} C_DIS
LIN {X -0.197,Y -572.537,Z 985.144,A 0.000,B 0.000,C 90.000,E1 61.897} C_DIS
LIN {X 0.041,Y -572.796,Z 985.136,A 0.000,B 0.000,C 90.000,E1 60.511} C_DIS
LIN {X -0.008,Y -573.005,Z 985.129,A 0.000,B 0.000,C 90.000,E1 59.154} C_DIS
LIN {X 0.037,Y -573.189,Z 985.121,A 0.000,B 0.000,C 90.000,E1 57.788} C_DIS
LIN {X 0.093,Y -573.302,Z 985.114,A 0.000,B 0.000,C 90.000,E1 56.421} C_DIS
LIN {X 0.146,Y -573.327,Z 985.106,A 0.000,B 0.000,C 90.000,E1 55.055} C_DIS
LIN {X 0.054,Y -573.070,Z 985.098,A 0.000,B 0.000,C 90.000,E1 53.703} C_DIS
LIN {X -0.183,Y -572.695,Z 985.092,A 0.000,B 0.000,C 90.000,E1 52.637} C_DIS
LIN {X -0.078,Y -572.111,Z 985.086,A 0.000,B 0.000,C 90.000,E1 51.537} C_DIS
LIN {X 0.022,Y -571.318,Z 985.080,A 0.000,B 0.000,C 90.000,E1 50.436} C_DIS
LIN {X -0.024,Y -570.652,Z 985.076,A 0.000,B 0.000,C 90.000,E1 49.622} C_DIS
LIN {X -0.011,Y -569.496,Z 985.070,A 0.000,B 0.000,C 90.000,E1 48.528} C_DIS
LIN {X -0.197,Y -568.857,Z 985.067,A 0.000,B 0.000,C 90.000,E1 48.000} C_DIS
LIN {X 0.106,Y -567.710,Z 985.062,A 0.000,B 0.000,C 90.000,E1 47.148} C_DIS
LIN {X 0.082,Y -565.830,Z 985.056,A 0.000,B 0.000,C 90.000,E1 46.053} C_DIS
LIN {X -0.059,Y -564.233,Z 985.051,A 0.000,B 0.000,C 90.000,E1 45.243} C_DIS
LIN {X 0.259,Y -561.875,Z 985.045,A 0.000,B 0.000,C 90.000,E1 44.109} C_DIS
LIN {X 0.073,Y -559.702,Z 985.041,A 0.000,B 0.000,C 90.000,E1 43.299} C_DIS
LIN {X -0.182,Y -558.151,Z 985.038,A 0.000,B 0.000,C 90.000,E1 42.771} C_DIS
LIN {X 0.003,Y -555.538,Z 985.033,A 0.000,B 0.000,C 90.000,E1 41.919} C_DIS
LIN {X 0.092,Y -553.657,Z 985.030,A 0.000,B 0.000,C 90.000,E1 41.353} C_DIS
LIN {X -0.140,Y -550.419,Z 985.025,A 0.000,B 0.000,C 90.000,E1 40.539} C_DIS
LIN {X 0.173,Y -547.519,Z 985.021,A 0.000,B 0.000,C 90.000,E1 39.806} C_DIS
LIN {X -0.158,Y -545.028,Z 985.018,A 0.000,B 0.000,C 90.000,E1 39.277} C_DIS
LIN {X 0.103,Y -541.661,Z 985.014,A 0.000,B 0.000,C 90.000,E1 38.543} C_DIS
LIN {X -0.084,Y -536.622,Z 985.009,A 0.000,B 0.000,C 90.000,E1 37.569} C_DIS
LIN {X -0.074,Y -531.986,Z 985.004,A 0.000,B 0.000,C 90.000,E1 36.710} C_DIS
LIN {X 0.313,Y -527.187,Z 984.999,A 0.000,B 0.000,C 90.000,E1 35.804} C_DIS
LIN {X -0.125,Y -520.175,Z 984.993,A 0.000,B 0.000,C 90.000,E1 34.692} C_DIS
LIN {X -0.046,Y -513.412,Z 984.987,A 0.000,B 0.000,C 90.000,E1 33.658} C_DIS
LIN {X 0.036,Y -508.182,Z 984.983,A 0.000,B 0.000,C 90.000,E1 32.911} C_DIS
LIN {X -0.163,Y -503.700,Z 984.980,A 0.000,B 0.000,C 90.000,E1 32.339} C_DIS
LIN {X -0.044,Y -500.229,Z 984.977,A 0.000,B 0.000,C 90.000,E1 31.878} C_DIS
LIN {X 0.114,Y -495.167,Z 984.974,A 0.000,B 0.000,C 90.000,E1 31.258} C_DIS
LIN {X 0.049,Y -489.745,Z 984.970,A 0.000,B 0.000,C 90.000,E1 30.669} C_DIS
LIN {X 0.085,Y -482.803,Z 984.966,A 0.000,B 0.000,C 90.000,E1 29.951} C_DIS
LIN {X -0.018,Y -474.262,Z 984.962,A 0.000,B 0.000,C 90.000,E1 29.127} C_DIS
LIN {X 0.076,Y -464.036,Z 984.956,A 0.000,B 0.000,C 90.000,E1 28.153} C_DIS
LIN {X -0.188,Y -453.620,Z 984.951,A 0.000,B 0.000,C 90.000,E1 27.257} C_DIS
LIN {X 0.073,Y -441.388,Z 984.946,A 0.000,B 0.000,C 90.000,E1 26.181} C_DIS
LIN {X 0.103,Y -423.460,Z 984.937,A 0.000,B 0.000,C 90.000,E1 24.591} C_DIS
LIN {X -0.121,Y -410.158,Z 984.930,A 0.000,B 0.000,C 90.000,E1 23.334} C_DIS
LIN {X 0.131,Y -401.418,Z 984.924,A 0.000,B 0.000,C 90.000,E1 22.386} C_DIS
LIN {X -0.227,Y -396.507,Z 984.921,A 0.000,B 0.000,C 90.000,E1 21.844} C_DIS
LIN {X -0.038,Y -393.743,Z 984.919,A 0.000,B 0.000,C 90.000,E1 21.408} C_DIS
LIN {X -0.005,Y -392.726,Z 984.918,A 0.000,B 0.000,C 90.000,E1 21.227} C_DIS
LIN {X -0.162,Y -391.263,Z 984.916,A 0.000,B 0.000,C 90.000,E1 20.918} C_DIS
LIN {X 0.130,Y -390.106,Z 984.912,A 0.000,B 0.000,C 90.000,E1 20.120} C_DIS
LIN {X -0.174,Y -389.978,Z 984.909,A 0.000,B 0.000,C 90.000,E1 19.631} C_DIS
LIN {X 0.082,Y -391.620,Z 984.897,A 0.000,B 0.000,C 90.000,E1 17.457} C_DIS
LIN {X -0.170,Y -394.339,Z 984.883,A 0.000,B 0.000,C 90.000,E1 15.009} C_DIS
LIN {X -0.135,Y -398.406,Z 984.866,A 0.000,B 0.000,C 90.000,E1 11.827} C_DIS
LIN {X 0.208,Y -403.468,Z 984.848,A 0.000,B 0.000,C 90.000,E1 8.624} C_DIS
LIN {X 0.147,Y -408.665,Z 984.833,A 0.000,B 0.000,C 90.000,E1 5.853} C_DIS
LIN {X 0.177,Y -415.233,Z 984.815,A 0.000,B 0.000,C 90.000,E1 2.751} C_DIS
LIN {X -0.169,Y -418.254,Z 984.808,A 0.000,B 0.000,C 90.000,E1 1.432} C_DIS
LIN {X -0.135,Y -419.668,Z 984.805,A 0.000,B 0.000,C 90.000,E1 0.917} C_DIS
LIN {X -0.086,Y -422.594,Z 984.801,A 0.000,B 0.000,C 90.000,E1 0.172} C_DIS
LIN {X 0.080,Y -424.106,Z 984.799,A 0.000,B 0.000,C 90.000,E1 359.885} C_DIS
LIN {X -0.023,Y -428.423,Z 984.797,A 0.000,B 0.000,C 90.000,E1 359.370} C_DIS
LIN {X 0.212,Y -429.309,Z 984.796,A 0.000,B 0.000,C 90.000,E1 359.255} C_DIS
LIN {X 0.164,Y -434.069,Z 984.794,A 0.000,B 0.000,C 90.000,E1 358.912} C_DIS
LIN {X 0.210,Y -448.375,Z 984.790,A 0.000,B 0.000,C 90.000,E1 358.108} C_DIS
LIN {X -0.174,Y -461.659,Z 984.786,A 0.000,B 0.000,C 90.000,E1 357.421} C_DIS
LIN {X -0.050,Y -471.789,Z 984.782,A 0.000,B 0.000,C 90.000,E1 356.846} C_DIS
LIN {X 0.069,Y -486.706,Z 984.778,A 0.000,B 0.000,C 90.000,E1 355.988} C_DIS
LIN {X 0.111,Y -496.542,Z 984.775,A 0.000,B 0.000,C 90.000,E1 355.412} C_DIS
LIN {X 0.031,Y -506.160,Z 984.771,A 0.000,B 0.000,C 90.000,E1 354.837} C_DIS
LIN {X 0.188,Y -513.979,Z 984.769,A 0.000,B 0.000,C 90.000,E1 354.318} C_DIS
LIN {X 0.183,Y -523.222,Z 984.765,A 0.000,B 0.000,C 90.000,E1 353.685} C_DIS
LIN {X -0.008,Y -531.838,Z 984.761,A 0.000,B 0.000,C 90.000,E1 353.053} C_DIS
LIN {X -0.029,Y -538.957,Z 984.758,A 0.000,B 0.000,C 90.000,E1 352.470} C_DIS
LIN {X 0.167,Y -546.691,Z 984.754,A 0.000,B 0.000,C 90.000,E1 351.724} C_DIS
LIN {X 0.190,Y -551.907,Z 984.751,A 0.000,B 0.000,C 90.000,E1 351.197} C_DIS
LIN {X -0.060,Y -556.861,Z 984.748,A 0.000,B 0.000,C 90.000,E1 350.679} C_DIS
LIN {X 0.213,Y -561.477,Z 984.745,A 0.000,B 0.000,C 90.000,E1 350.095} C_DIS
LIN {X -0.158,Y -566.620,Z 984.741,A 0.000,B 0.000,C 90.000,E1 349.454} C_DIS
LIN {X 0.193,Y -570.465,Z 984.738,A 0.000,B 0.000,C 90.000,E1 348.870} C_DIS
LIN {X 0.213,Y -575.675,Z 984.734,A 0.000,B 0.000,C 90.000,E1 348.049} C_DIS
LIN {X -0.168,Y -579.573,Z 984.730,A 0.000,B 0.000,C 90.000,E1 347.409} C_DIS
LIN {X -0.157,Y -584.776,Z 984.725,A 0.000,B 0.000,C 90.000,E1 346.464} C_DIS
LIN {X -0.081,Y -589.551,Z 984.720,A 0.000,B 0.000,C 90.000,E1 345.519} C_DIS
LIN {X -0.020,Y -594.806,Z 984.714,A 0.000,B 0.000,C 90.000,E1 344.448} C_DIS
LIN {X -0.230,Y -601.509,Z 984.706,A 0.000,B 0.000,C 90.000,E1 343.015} C_DIS
LIN {X -0.020,Y -605.947,Z 984.700,A 0.000,B 0.000,C 90.000,E1 341.945} C_DIS
LIN {X -0.142,Y -610.245,Z 984.694,A 0.000,B 0.000,C 90.000,E1 340.913} C_DIS
LIN {X -0.207,Y -614.198,Z 984.688,A 0.000,B 0.000,C 90.000,E1 339.880} C_DIS
LIN {X 0.033,Y -616.925,Z 984.684,A 0.000,B 0.000,C 90.000,E1 339.082} C_DIS
LIN {X 0.051,Y -620.374,Z 984.678,A 0.000,B 0.000,C 90.000,E1 338.050} C_DIS
LIN {X -0.233,Y -624.433,Z 984.671,A 0.000,B 0.000,C 90.000,E1 336.794} C_DIS
LIN {X 0.127,Y -628.089,Z 984.664,A 0.000,B 0.000,C 90.000,E1 335.485} C_DIS
LIN {X 0.216,Y -630.829,Z 984.658,A 0.000,B 0.000,C 90.000,E1 334.460} C_DIS
LIN {X 0.066,Y -633.307,Z 984.653,A 0.000,B 0.000,C 90.000,E1 333.461} C_DIS
LIN {X 0.181,Y -635.040,Z 984.648,A 0.000,B 0.000,C 90.000,E1 332.692} C_DIS
LIN {X 0.198,Y -638.169,Z 984.640,A 0.000,B 0.000,C 90.000,E1 331.179} C_DIS
LIN {X -0.146,Y -640.101,Z 984.634,A 0.000,B 0.000,C 90.000,E1 330.205} C_DIS
LIN {X -0.149,Y -641.964,Z 984.629,A 0.000,B 0.000,C 90.000,E1 329.203} C_DIS
LIN {X 0.275,Y -643.921,Z 984.622,A 0.000,B 0.000,C 90.000,E1 327.916} C_DIS
LIN {X -0.219,Y -645.333,Z 984.616,A 0.000,B 0.000,C 90.000,E1 326.962} C_DIS
LIN {X 0.257,Y -646.861,Z 984.609,A 0.000,B 0.000,C 90.000,E1 325.674} C_DIS
LIN {X -0.318,Y -648.014,Z 984.603,A 0.000,B 0.000,C 90.000,E1 324.482} C_DIS
LIN {X 0.028,Y -648.911,Z 984.596,A 0.000,B 0.000,C 90.000,E1 323.210} C_DIS
LIN {X -0.133,Y -649.480,Z 984.589,A 0.000,B 0.000,C 90.000,E1 321.984} C_DIS
LIN {X 0.121,Y -650.084,Z 984.582,A 0.000,B 0.000,C 90.000,E1 320.723} C_DIS
LIN {X -0.096,Y -650.695,Z 984.574,A 0.000,B 0.000,C 90.000,E1 319.256} C_DIS
LIN {X -0.053,Y -652.044,Z 984.561,A 0.000,B 0.000,C 90.000,E1 317.025} C_DIS
LIN {X -0.289,Y -652.935,Z 984.554,A 0.000,B 0.000,C 90.000,E1 315.810} C_DIS
LIN {X 0.383,Y -654.040,Z 984.546,A 0.000,B 0.000,C 90.000,E1 314.271} C_DIS
LIN {X -0.344,Y -655.406,Z 984.537,A 0.000,B 0.000,C 90.000,E1 312.609} C_DIS
LIN {X -0.014,Y -656.123,Z 984.531,A 0.000,B 0.000,C 90.000,E1 311.595} C_DIS
LIN {X -0.149,Y -656.976,Z 984.524,A 0.000,B 0.000,C 90.000,E1 310.378} C_DIS
LIN {X 0.231,Y -657.683,Z 984.517,A 0.000,B 0.000,C 90.000,E1 309.116} C_DIS
LIN {X -0.286,Y -658.495,Z 984.508,A 0.000,B 0.000,C 90.000,E1 307.443} C_DIS
LIN {X 0.157,Y -658.852,Z 984.503,A 0.000,B 0.000,C 90.000,E1 306.423} C_DIS
LIN {X -0.110,Y -659.165,Z 984.492,A 0.000,B 0.000,C 90.000,E1 304.485} C_DIS
LIN {X 0.367,Y -660.415,Z 984.474,A 0.000,B 0.000,C 90.000,E1 301.258} C_DIS
LIN {X 0.239,Y -665.224,Z 984.449,A 0.000,B 0.000,C 90.000,E1 296.873} C_DIS
LIN {X -0.190,Y -668.040,Z 984.440,A 0.000,B 0.000,C 90.000,E1 295.207} C_DIS
LIN {X 0.322,Y -669.988,Z 984.433,A 0.000,B 0.000,C 90.000,E1 293.951} C_DIS
LIN {X -0.177,Y -671.388,Z 984.428,A 0.000,B 0.000,C 90.000,E1 293.025} C_DIS
LIN {X 0.150,Y -671.842,Z 984.425,A 0.000,B 0.000,C 90.000,E1 292.514} C_DIS
LIN {X 0.221,Y -671.961,Z 984.422,A 0.000,B 0.000,C 90.000,E1 292.025} C_DIS
LIN {X 0.134,Y -671.927,Z 984.421,A 0.000,B 0.000,C 90.000,E1 291.791} C_DIS
LIN {X -0.168,Y -671.240,Z 984.419,A 0.000,B 0.000,C 90.000,E1 291.334} C_DIS
LIN {X -0.254,Y -670.710,Z 984.417,A 0.000,B 0.000,C 90.000,E1 291.099} C_DIS
LIN {X -0.176,Y -670.187,Z 984.417,A 0.000,B 0.000,C 90.000,E1 290.972} C_DIS
LIN {X -0.114,Y -666.678,Z 984.414,A 0.000,B 0.000,C 90.000,E1 290.482} C_DIS
LIN {X -0.043,Y -665.669,Z 984.413,A 0.000,B 0.000,C 90.000,E1 290.355} C_DIS
LIN {X -0.205,Y -664.311,Z 984.412,A 0.000,B 0.000,C 90.000,E1 290.248} C_DIS
LIN {X -0.036,Y -658.271,Z 984.410,A 0.000,B 0.000,C 90.000,E1 289.812} C_DIS
LIN {X -0.109,Y -651.973,Z 984.408,A 0.000,B 0.000,C 90.000,E1 289.450} C_DIS
LIN {X 0.173,Y -647.801,Z 984.406,A 0.000,B 0.000,C 90.000,E1 289.141} C_DIS
LIN {X -0.020,Y -647.228,Z 984.406,A 0.000,B 0.000,C 90.000,E1 289.087} C_DIS
LIN {X -0.055,Y -647.222,Z 984.406,A 0.000,B 0.000,C 90.000,E1 289.087} C_DIS
LIN {X -0.039,Y -647.583,Z 984.405,A 0.000,B 0.000,C 90.000,E1 288.906} C_DIS
LIN {X -0.009,Y -647.985,Z 984.404,A 0.000,B 0.000,C 90.000,E1 288.779} C_DIS
LIN {X -0.094,Y -650.453,Z 984.402,A 0.000,B 0.000,C 90.000,E1 288.290} C_DIS
LIN {X 0.030,Y -655.608,Z 984.397,A 0.000,B 0.000,C 90.000,E1 287.457} C_DIS
LIN {X -0.163,Y -659.125,Z 984.394,A 0.000,B 0.000,C 90.000,E1 286.858} C_DIS
LIN {X -0.331,Y -662.326,Z 984.390,A 0.000,B 0.000,C 90.000,E1 286.260} C_DIS
LIN {X 0.118,Y -664.383,Z 984.388,A 0.000,B 0.000,C 90.000,E1 285.733} C_DIS
LIN {X 0.208,Y -665.279,Z 984.386,A 0.000,B 0.000,C 90.000,E1 285.481} C_DIS
LIN {X 0.037,Y -666.764,Z 984.383,A 0.000,B 0.000,C 90.000,E1 285.009} C_DIS
LIN {X -0.200,Y -668.465,Z 984.379,A 0.000,B 0.000,C 90.000,E1 284.300} C_DIS
LIN {X 0.231,Y -669.578,Z 984.375,A 0.000,B 0.000,C 90.000,E1 283.536} C_DIS
LIN {X 0.091,Y -670.173,Z 984.373,A 0.000,B 0.000,C 90.000,E1 283.063} C_DIS
LIN {X -0.045,Y -670.547,Z 984.370,A 0.000,B 0.000,C 90.000,E1 282.591} C_DIS
LIN {X -0.183,Y -670.722,Z 984.367,A 0.000,B 0.000,C 90.000,E1 282.119} C_DIS
LIN {X 0.134,Y -670.591,Z 984.363,A 0.000,B 0.000,C 90.000,E1 281.366} C_DIS
LIN {X -0.005,Y -670.358,Z 984.361,A 0.000,B 0.000,C 90.000,E1 280.894} C_DIS
LIN {X -0.343,Y -669.479,Z 984.357,A 0.000,B 0.000,C 90.000,E1 280.197} C_DIS
LIN {X 0.163,Y -668.663,Z 984.354,A 0.000,B 0.000,C 90.000,E1 279.670} C_DIS
LIN {X -0.107,Y -667.529,Z 984.351,A 0.000,B 0.000,C 90.000,E1 279.208} C_DIS
LIN {X 0.278,Y -666.115,Z 984.348,A 0.000,B 0.000,C 90.000,E1 278.690} C_DIS
LIN {X 0.094,Y -664.344,Z 984.346,A 0.000,B 0.000,C 90.000,E1 278.219} C_DIS
LIN {X -0.198,Y -662.332,Z 984.343,A 0.000,B 0.000,C 90.000,E1 277.757} C_DIS
LIN {X 0.252,Y -660.521,Z 984.341,A 0.000,B 0.000,C 90.000,E1 277.352} C_DIS
LIN {X 0.036,Y -658.523,Z 984.339,A 0.000,B 0.000,C 90.000,E1 277.004} C_DIS
LIN {X 0.356,Y -655.426,Z 984.336,A 0.000,B 0.000,C 90.000,E1 276.486} C_DIS
LIN {X -0.104,Y -650.868,Z 984.333,A 0.000,B 0.000,C 90.000,E1 275.910} C_DIS
LIN {X 0.051,Y -645.650,Z 984.329,A 0.000,B 0.000,C 90.000,E1 275.277} C_DIS
LIN {X 0.280,Y -641.104,Z 984.327,A 0.000,B 0.000,C 90.000,E1 274.759} C_DIS
LIN {X -0.170,Y -636.120,Z 984.324,A 0.000,B 0.000,C 90.000,E1 274.302} C_DIS
LIN {X 0.276,Y -630.918,Z 984.321,A 0.000,B 0.000,C 90.000,E1 273.784} C_DIS
LIN {X 0.257,Y -623.928,Z 984.318,A 0.000,B 0.000,C 90.000,E1 273.212} C_DIS
LIN {X -0.076,Y -618.107,Z 984.316,A 0.000,B 0.000,C 90.000,E1 272.808} C_DIS
LIN {X 0.038,Y -610.485,Z 984.313,A 0.000,B 0.000,C 90.000,E1 272.293} C_DIS
LIN {X 0.044,Y -605.628,Z 984.311,A 0.000,B 0.000,C 90.000,E1 272.007} C_DIS
LIN {X -0.258,Y -597.236,Z 984.309,A 0.000,B 0.000,C 90.000,E1 271.604} C_DIS
LIN {X 0.117,Y -590.068,Z 984.307,A 0.000,B 0.000,C 90.000,E1 271.260} C_DIS
LIN {X -0.199,Y -584.830,Z 984.306,A 0.000,B 0.000,C 90.000,E1 271.088} C_DIS
LIN {X -0.266,Y -577.264,Z 984.305,A 0.000,B 0.000,C 90.000,E1 270.859} C_DIS
LIN {X 0.011,Y -571.529,Z 984.304,A 0.000,B 0.000,C 90.000,E1 270.688} C_DIS
LIN {X -0.096,Y -565.412,Z 984.303,A 0.000,B 0.000,C 90.000,E1 270.573} C_DIS
LIN {X -0.141,Y -560.072,Z 984.303,A 0.000,B 0.000,C 90.000,E1 270.516} C_DIS
LIN {X 0.223,Y -557.820,Z 984.303,A 0.000,B 0.000,C 90.000,E1 270.458} C_DIS
LIN {X 0.186,Y -545.052,Z 984.303,A 0.000,B 0.000,C 90.000,E1 270.458} C_DIS
LIN {X 0.106,Y -542.865,Z 984.302,A 0.000,B 0.000,C 90.000,E1 270.344} C_DIS
LIN {X 0.052,Y -542.815,Z 984.302,A 0.000,B 0.000,C 90.000,E1 270.344} C_DIS
LIN {X -0.233,Y -540.905,Z 984.287,A 0.000,B 0.000,C 90.000,E1 267.764} C_DIS
LIN {X -0.047,Y -539.471,Z 984.276,A 0.000,B 0.000,C 90.000,E1 265.755} C_DIS
LIN {X 0.082,Y -538.418,Z 984.269,A 0.000,B 0.000,C 90.000,E1 264.318} C_DIS
LIN {X 0.189,Y -537.441,Z 984.262,A 0.000,B 0.000,C 90.000,E1 263.166} C_DIS
LIN {X -0.149,Y -535.777,Z 984.253,A 0.000,B 0.000,C 90.000,E1 261.489} C_DIS
LIN {X -0.016,Y -534.620,Z 984.246,A 0.000,B 0.000,C 90.000,E1 260.330} C_DIS
LIN {X 0.241,Y -533.096,Z 984.238,A 0.000,B 0.000,C 90.000,E1 258.870} C_DIS
LIN {X -0.006,Y -531.237,Z 984.229,A 0.000,B 0.000,C 90.000,E1 257.173} C_DIS
LIN {X 0.012,Y -528.459,Z 984.216,A 0.000,B 0.000,C 90.000,E1 254.866} C_DIS
LIN {X 0.082,Y -526.350,Z 984.205,A 0.000,B 0.000,C 90.000,E1 252.834} C_DIS
LIN {X -0.075,Y -524.994,Z 984.198,A 0.000,B 0.000,C 90.000,E1 251.692} C_DIS
LIN {X -0.256,Y -523.560,Z 984.192,A 0.000,B 0.000,C 90.000,E1 250.550} C_DIS
LIN {X -0.131,Y -521.715,Z 984.184,A 0.000,B 0.000,C 90.000,E1 249.082} C_DIS
LIN {X 0.102,Y -519.453,Z 984.174,A 0.000,B 0.000,C 90.000,E1 247.305} C_DIS
LIN {X 0.054,Y -518.250,Z 984.169,A 0.000,B 0.000,C 90.000,E1 246.433} C_DIS
LIN {X 0.004,Y -516.083,Z 984.161,A 0.000,B 0.000,C 90.000,E1 244.973} C_DIS
LIN {X -0.081,Y -513.718,Z 984.153,A 0.000,B 0.000,C 90.000,E1 243.512} C_DIS
LIN {X -0.319,Y -511.894,Z 984.146,A 0.000,B 0.000,C 90.000,E1 242.359} C_DIS
LIN {X 0.102,Y -509.957,Z 984.140,A 0.000,B 0.000,C 90.000,E1 241.129} C_DIS
LIN {X -0.034,Y -508.471,Z 984.135,A 0.000,B 0.000,C 90.000,E1 240.255} C_DIS
LIN {X 0.208,Y -505.774,Z 984.127,A 0.000,B 0.000,C 90.000,E1 238.742} C_DIS
LIN {X 0.032,Y -504.008,Z 984.122,A 0.000,B 0.000,C 90.000,E1 237.867} C_DIS
END
